  STRUCT
   STAT0 : WORD ;
   STAT1 : WORD ;
   STAT2 : WORD ;
   STAT3 : WORD ;
   STAT4 : WORD ;
   STAT5 : WORD ;
   STAT6 : WORD ;
   STAT7 : WORD ;
   STAT8 : WORD ;
   STAT9 : WORD ;
   STAT10 : WORD ;
   STAT11 : WORD ;
   STAT12 : WORD ;
   STAT13 : WORD ;
   STAT14 : WORD ;
   STAT15 : WORD ;
   STAT16 : INT ;
   STAT17 : INT ;
   STAT18 : INT ;
   STAT19 : INT ;
   STAT20 : ARRAY  [1 .. 6 ] OF BYTE ;
   STAT21 : ARRAY  [1 .. 6 ] OF BYTE ;
   STAT22 : ARRAY  [1 .. 40 ] OF BOOL  := FALSE;
   STAT23 : ARRAY  [1 .. 40 ] OF BOOL  := FALSE;
   STAT24 : WORD ;
   STAT25 : WORD ;
   STAT26 : WORD ;
   STAT27 : WORD ;
   STAT28 : WORD ;
   STAT29 : WORD ;
   STAT30 : WORD ;
   STAT31 : ARRAY  [1 .. 7 ] OF WORD ;
   STAT32 : INT ;
   STAT33 : INT ;
   STAT34 : INT ;
   STAT35 : INT ;
   STAT36 : ARRAY  [1 .. 500 ] OF WORD ;
   STAT37 : ARRAY  [1 .. 16 ] OF BYTE ;
   STAT38 : ARRAY  [1 .. 4 ] OF BYTE ;
   STAT39 : ARRAY  [1 .. 16 ] OF BYTE ;
  END_STRUCT ;
BEGIN
   STAT0 := W#16#0;
   STAT1 := W#16#0;
   STAT2 := W#16#0;
   STAT3 := W#16#0;
   STAT4 := W#16#0;
   STAT5 := W#16#0;
   STAT6 := W#16#0;
   STAT7 := W#16#0;
   STAT8 := W#16#1;
   STAT9 := W#16#9515;
   STAT10 := W#16#2212;
   STAT11 := W#16#8004;
   STAT12 := W#16#1644;
   STAT13 := W#16#0;
   STAT14 := W#16#0;
   STAT15 := W#16#0;
   STAT16 := 0;
   STAT17 := 8;
   STAT18 := 3;
   STAT19 := 0;
   STAT20[1] := B#16#0;
   STAT20[2] := B#16#0;
   STAT20[3] := B#16#0;
   STAT20[4] := B#16#0;
   STAT20[5] := B#16#0;
   STAT20[6] := B#16#0;
   STAT21[1] := B#16#0;
   STAT21[2] := B#16#0;
   STAT21[3] := B#16#0;
   STAT21[4] := B#16#0;
   STAT21[5] := B#16#0;
   STAT21[6] := B#16#0;
   STAT22[1] := FALSE;
   STAT22[2] := FALSE;
   STAT22[3] := TRUE;
   STAT22[4] := FALSE;
   STAT22[5] := FALSE;
   STAT22[6] := FALSE;
   STAT22[7] := FALSE;
   STAT22[8] := TRUE;
   STAT22[9] := FALSE;
   STAT22[10] := FALSE;
   STAT22[11] := FALSE;
   STAT22[12] := FALSE;
   STAT22[13] := FALSE;
   STAT22[14] := FALSE;
   STAT22[15] := FALSE;
   STAT22[16] := FALSE;
   STAT22[17] := FALSE;
   STAT22[18] := FALSE;
   STAT22[19] := FALSE;
   STAT22[20] := FALSE;
   STAT22[21] := FALSE;
   STAT22[22] := FALSE;
   STAT22[23] := FALSE;
   STAT22[24] := FALSE;
   STAT22[25] := FALSE;
   STAT22[26] := FALSE;
   STAT22[27] := FALSE;
   STAT22[28] := FALSE;
   STAT22[29] := FALSE;
   STAT22[30] := FALSE;
   STAT22[31] := FALSE;
   STAT22[32] := FALSE;
   STAT22[33] := FALSE;
   STAT22[34] := FALSE;
   STAT22[35] := FALSE;
   STAT22[36] := FALSE;
   STAT22[37] := FALSE;
   STAT22[38] := FALSE;
   STAT22[39] := FALSE;
   STAT22[40] := FALSE;
   STAT23[1] := FALSE;
   STAT23[2] := FALSE;
   STAT23[3] := FALSE;
   STAT23[4] := FALSE;
   STAT23[5] := FALSE;
   STAT23[6] := TRUE;
   STAT23[7] := FALSE;
   STAT23[8] := FALSE;
   STAT23[9] := FALSE;
   STAT23[10] := FALSE;
   STAT23[11] := FALSE;
   STAT23[12] := FALSE;
   STAT23[13] := FALSE;
   STAT23[14] := FALSE;
   STAT23[15] := FALSE;
   STAT23[16] := FALSE;
   STAT23[17] := FALSE;
   STAT23[18] := FALSE;
   STAT23[19] := FALSE;
   STAT23[20] := FALSE;
   STAT23[21] := FALSE;
   STAT23[22] := FALSE;
   STAT23[23] := FALSE;
   STAT23[24] := FALSE;
   STAT23[25] := TRUE;
   STAT23[26] := FALSE;
   STAT23[27] := FALSE;
   STAT23[28] := FALSE;
   STAT23[29] := FALSE;
   STAT23[30] := FALSE;
   STAT23[31] := FALSE;
   STAT23[32] := FALSE;
   STAT23[33] := FALSE;
   STAT23[34] := FALSE;
   STAT23[35] := FALSE;
   STAT23[36] := FALSE;
   STAT23[37] := FALSE;
   STAT23[38] := FALSE;
   STAT23[39] := FALSE;
   STAT23[40] := FALSE;
   STAT24 := W#16#0;
   STAT25 := W#16#0;
   STAT26 := W#16#0;
   STAT27 := W#16#0;
   STAT28 := W#16#0;
   STAT29 := W#16#0;
   STAT30 := W#16#0;
   STAT31[1] := W#16#0;
   STAT31[2] := W#16#0;
   STAT31[3] := W#16#0;
   STAT31[4] := W#16#0;
   STAT31[5] := W#16#0;
   STAT31[6] := W#16#0;
   STAT31[7] := W#16#0;
   STAT32 := 100;
   STAT33 := 90;
   STAT34 := 80;
   STAT35 := 0;
   STAT36[1] := W#16#600;
   STAT36[2] := W#16#808;
   STAT36[3] := W#16#2930;
   STAT36[4] := W#16#64;
   STAT36[5] := W#16#1;
   STAT36[6] := W#16#600;
   STAT36[7] := W#16#1223;
   STAT36[8] := W#16#4457;
   STAT36[9] := W#16#64;
   STAT36[10] := W#16#9515;
   STAT36[11] := W#16#600;
   STAT36[12] := W#16#908;
   STAT36[13] := W#16#2517;
   STAT36[14] := W#16#64;
   STAT36[15] := W#16#341;
   STAT36[16] := W#16#600;
   STAT36[17] := W#16#522;
   STAT36[18] := W#16#356;
   STAT36[19] := W#16#64;
   STAT36[20] := W#16#8579;
   STAT36[21] := W#16#500;
   STAT36[22] := W#16#1220;
   STAT36[23] := W#16#3131;
   STAT36[24] := W#16#0;
   STAT36[25] := W#16#0;
   STAT36[26] := W#16#0;
   STAT36[27] := W#16#0;
   STAT36[28] := W#16#0;
   STAT36[29] := W#16#0;
   STAT36[30] := W#16#0;
   STAT36[31] := W#16#0;
   STAT36[32] := W#16#0;
   STAT36[33] := W#16#0;
   STAT36[34] := W#16#0;
   STAT36[35] := W#16#0;
   STAT36[36] := W#16#0;
   STAT36[37] := W#16#0;
   STAT36[38] := W#16#0;
   STAT36[39] := W#16#0;
   STAT36[40] := W#16#0;
   STAT36[41] := W#16#0;
   STAT36[42] := W#16#0;
   STAT36[43] := W#16#0;
   STAT36[44] := W#16#0;
   STAT36[45] := W#16#0;
   STAT36[46] := W#16#0;
   STAT36[47] := W#16#0;
   STAT36[48] := W#16#0;
   STAT36[49] := W#16#0;
   STAT36[50] := W#16#0;
   STAT36[51] := W#16#0;
   STAT36[52] := W#16#0;
   STAT36[53] := W#16#0;
   STAT36[54] := W#16#0;
   STAT36[55] := W#16#0;
   STAT36[56] := W#16#0;
   STAT36[57] := W#16#0;
   STAT36[58] := W#16#0;
   STAT36[59] := W#16#0;
   STAT36[60] := W#16#0;
   STAT36[61] := W#16#0;
   STAT36[62] := W#16#0;
   STAT36[63] := W#16#0;
   STAT36[64] := W#16#0;
   STAT36[65] := W#16#0;
   STAT36[66] := W#16#0;
   STAT36[67] := W#16#0;
   STAT36[68] := W#16#0;
   STAT36[69] := W#16#0;
   STAT36[70] := W#16#0;
   STAT36[71] := W#16#0;
   STAT36[72] := W#16#0;
   STAT36[73] := W#16#0;
   STAT36[74] := W#16#0;
   STAT36[75] := W#16#0;
   STAT36[76] := W#16#0;
   STAT36[77] := W#16#0;
   STAT36[78] := W#16#0;
   STAT36[79] := W#16#0;
   STAT36[80] := W#16#0;
   STAT36[81] := W#16#0;
   STAT36[82] := W#16#0;
   STAT36[83] := W#16#0;
   STAT36[84] := W#16#0;
   STAT36[85] := W#16#0;
   STAT36[86] := W#16#0;
   STAT36[87] := W#16#0;
   STAT36[88] := W#16#0;
   STAT36[89] := W#16#0;
   STAT36[90] := W#16#0;
   STAT36[91] := W#16#0;
   STAT36[92] := W#16#0;
   STAT36[93] := W#16#0;
   STAT36[94] := W#16#0;
   STAT36[95] := W#16#0;
   STAT36[96] := W#16#0;
   STAT36[97] := W#16#0;
   STAT36[98] := W#16#0;
   STAT36[99] := W#16#0;
   STAT36[100] := W#16#0;
   STAT36[101] := W#16#0;
   STAT36[102] := W#16#0;
   STAT36[103] := W#16#0;
   STAT36[104] := W#16#0;
   STAT36[105] := W#16#0;
   STAT36[106] := W#16#0;
   STAT36[107] := W#16#0;
   STAT36[108] := W#16#0;
   STAT36[109] := W#16#0;
   STAT36[110] := W#16#0;
   STAT36[111] := W#16#0;
   STAT36[112] := W#16#0;
   STAT36[113] := W#16#0;
   STAT36[114] := W#16#0;
   STAT36[115] := W#16#0;
   STAT36[116] := W#16#0;
   STAT36[117] := W#16#0;
   STAT36[118] := W#16#0;
   STAT36[119] := W#16#0;
   STAT36[120] := W#16#0;
   STAT36[121] := W#16#0;
   STAT36[122] := W#16#0;
   STAT36[123] := W#16#0;
   STAT36[124] := W#16#0;
   STAT36[125] := W#16#0;
   STAT36[126] := W#16#0;
   STAT36[127] := W#16#0;
   STAT36[128] := W#16#0;
   STAT36[129] := W#16#0;
   STAT36[130] := W#16#0;
   STAT36[131] := W#16#0;
   STAT36[132] := W#16#0;
   STAT36[133] := W#16#0;
   STAT36[134] := W#16#0;
   STAT36[135] := W#16#0;
   STAT36[136] := W#16#0;
   STAT36[137] := W#16#0;
   STAT36[138] := W#16#0;
   STAT36[139] := W#16#0;
   STAT36[140] := W#16#0;
   STAT36[141] := W#16#0;
   STAT36[142] := W#16#0;
   STAT36[143] := W#16#0;
   STAT36[144] := W#16#0;
   STAT36[145] := W#16#0;
   STAT36[146] := W#16#0;
   STAT36[147] := W#16#0;
   STAT36[148] := W#16#0;
   STAT36[149] := W#16#0;
   STAT36[150] := W#16#0;
   STAT36[151] := W#16#0;
   STAT36[152] := W#16#0;
   STAT36[153] := W#16#0;
   STAT36[154] := W#16#0;
   STAT36[155] := W#16#0;
   STAT36[156] := W#16#0;
   STAT36[157] := W#16#0;
   STAT36[158] := W#16#0;
   STAT36[159] := W#16#0;
   STAT36[160] := W#16#0;
   STAT36[161] := W#16#0;
   STAT36[162] := W#16#0;
   STAT36[163] := W#16#0;
   STAT36[164] := W#16#0;
   STAT36[165] := W#16#0;
   STAT36[166] := W#16#0;
   STAT36[167] := W#16#0;
   STAT36[168] := W#16#0;
   STAT36[169] := W#16#0;
   STAT36[170] := W#16#0;
   STAT36[171] := W#16#0;
   STAT36[172] := W#16#0;
   STAT36[173] := W#16#0;
   STAT36[174] := W#16#0;
   STAT36[175] := W#16#0;
   STAT36[176] := W#16#0;
   STAT36[177] := W#16#0;
   STAT36[178] := W#16#0;
   STAT36[179] := W#16#0;
   STAT36[180] := W#16#0;
   STAT36[181] := W#16#0;
   STAT36[182] := W#16#0;
   STAT36[183] := W#16#0;
   STAT36[184] := W#16#0;
   STAT36[185] := W#16#0;
   STAT36[186] := W#16#0;
   STAT36[187] := W#16#0;
   STAT36[188] := W#16#0;
   STAT36[189] := W#16#0;
   STAT36[190] := W#16#0;
   STAT36[191] := W#16#0;
   STAT36[192] := W#16#0;
   STAT36[193] := W#16#0;
   STAT36[194] := W#16#0;
   STAT36[195] := W#16#0;
   STAT36[196] := W#16#0;
   STAT36[197] := W#16#0;
   STAT36[198] := W#16#0;
   STAT36[199] := W#16#0;
   STAT36[200] := W#16#0;
   STAT36[201] := W#16#0;
   STAT36[202] := W#16#0;
   STAT36[203] := W#16#0;
   STAT36[204] := W#16#0;
   STAT36[205] := W#16#0;
   STAT36[206] := W#16#0;
   STAT36[207] := W#16#0;
   STAT36[208] := W#16#0;
   STAT36[209] := W#16#0;
   STAT36[210] := W#16#0;
   STAT36[211] := W#16#0;
   STAT36[212] := W#16#0;
   STAT36[213] := W#16#0;
   STAT36[214] := W#16#0;
   STAT36[215] := W#16#0;
   STAT36[216] := W#16#0;
   STAT36[217] := W#16#0;
   STAT36[218] := W#16#0;
   STAT36[219] := W#16#0;
   STAT36[220] := W#16#0;
   STAT36[221] := W#16#0;
   STAT36[222] := W#16#0;
   STAT36[223] := W#16#0;
   STAT36[224] := W#16#0;
   STAT36[225] := W#16#0;
   STAT36[226] := W#16#0;
   STAT36[227] := W#16#0;
   STAT36[228] := W#16#0;
   STAT36[229] := W#16#0;
   STAT36[230] := W#16#0;
   STAT36[231] := W#16#0;
   STAT36[232] := W#16#0;
   STAT36[233] := W#16#0;
   STAT36[234] := W#16#0;
   STAT36[235] := W#16#0;
   STAT36[236] := W#16#0;
   STAT36[237] := W#16#0;
   STAT36[238] := W#16#0;
   STAT36[239] := W#16#0;
   STAT36[240] := W#16#0;
   STAT36[241] := W#16#0;
   STAT36[242] := W#16#0;
   STAT36[243] := W#16#0;
   STAT36[244] := W#16#0;
   STAT36[245] := W#16#0;
   STAT36[246] := W#16#0;
   STAT36[247] := W#16#0;
   STAT36[248] := W#16#0;
   STAT36[249] := W#16#0;
   STAT36[250] := W#16#0;
   STAT36[251] := W#16#0;
   STAT36[252] := W#16#0;
   STAT36[253] := W#16#0;
   STAT36[254] := W#16#0;
   STAT36[255] := W#16#0;
   STAT36[256] := W#16#0;
   STAT36[257] := W#16#0;
   STAT36[258] := W#16#0;
   STAT36[259] := W#16#0;
   STAT36[260] := W#16#0;
   STAT36[261] := W#16#0;
   STAT36[262] := W#16#0;
   STAT36[263] := W#16#0;
   STAT36[264] := W#16#0;
   STAT36[265] := W#16#0;
   STAT36[266] := W#16#0;
   STAT36[267] := W#16#0;
   STAT36[268] := W#16#0;
   STAT36[269] := W#16#0;
   STAT36[270] := W#16#0;
   STAT36[271] := W#16#0;
   STAT36[272] := W#16#0;
   STAT36[273] := W#16#0;
   STAT36[274] := W#16#0;
   STAT36[275] := W#16#0;
   STAT36[276] := W#16#0;
   STAT36[277] := W#16#0;
   STAT36[278] := W#16#0;
   STAT36[279] := W#16#0;
   STAT36[280] := W#16#0;
   STAT36[281] := W#16#0;
   STAT36[282] := W#16#0;
   STAT36[283] := W#16#0;
   STAT36[284] := W#16#0;
   STAT36[285] := W#16#0;
   STAT36[286] := W#16#0;
   STAT36[287] := W#16#0;
   STAT36[288] := W#16#0;
   STAT36[289] := W#16#0;
   STAT36[290] := W#16#0;
   STAT36[291] := W#16#0;
   STAT36[292] := W#16#0;
   STAT36[293] := W#16#0;
   STAT36[294] := W#16#0;
   STAT36[295] := W#16#0;
   STAT36[296] := W#16#0;
   STAT36[297] := W#16#0;
   STAT36[298] := W#16#0;
   STAT36[299] := W#16#0;
   STAT36[300] := W#16#0;
   STAT36[301] := W#16#0;
   STAT36[302] := W#16#0;
   STAT36[303] := W#16#0;
   STAT36[304] := W#16#0;
   STAT36[305] := W#16#0;
   STAT36[306] := W#16#0;
   STAT36[307] := W#16#0;
   STAT36[308] := W#16#0;
   STAT36[309] := W#16#0;
   STAT36[310] := W#16#0;
   STAT36[311] := W#16#0;
   STAT36[312] := W#16#0;
   STAT36[313] := W#16#0;
   STAT36[314] := W#16#0;
   STAT36[315] := W#16#0;
   STAT36[316] := W#16#0;
   STAT36[317] := W#16#0;
   STAT36[318] := W#16#0;
   STAT36[319] := W#16#0;
   STAT36[320] := W#16#0;
   STAT36[321] := W#16#0;
   STAT36[322] := W#16#0;
   STAT36[323] := W#16#0;
   STAT36[324] := W#16#0;
   STAT36[325] := W#16#0;
   STAT36[326] := W#16#0;
   STAT36[327] := W#16#0;
   STAT36[328] := W#16#0;
   STAT36[329] := W#16#0;
   STAT36[330] := W#16#0;
   STAT36[331] := W#16#0;
   STAT36[332] := W#16#0;
   STAT36[333] := W#16#0;
   STAT36[334] := W#16#0;
   STAT36[335] := W#16#0;
   STAT36[336] := W#16#0;
   STAT36[337] := W#16#0;
   STAT36[338] := W#16#0;
   STAT36[339] := W#16#0;
   STAT36[340] := W#16#0;
   STAT36[341] := W#16#0;
   STAT36[342] := W#16#0;
   STAT36[343] := W#16#0;
   STAT36[344] := W#16#0;
   STAT36[345] := W#16#0;
   STAT36[346] := W#16#0;
   STAT36[347] := W#16#0;
   STAT36[348] := W#16#0;
   STAT36[349] := W#16#0;
   STAT36[350] := W#16#0;
   STAT36[351] := W#16#0;
   STAT36[352] := W#16#0;
   STAT36[353] := W#16#0;
   STAT36[354] := W#16#0;
   STAT36[355] := W#16#0;
   STAT36[356] := W#16#0;
   STAT36[357] := W#16#0;
   STAT36[358] := W#16#0;
   STAT36[359] := W#16#0;
   STAT36[360] := W#16#0;
   STAT36[361] := W#16#0;
   STAT36[362] := W#16#0;
   STAT36[363] := W#16#0;
   STAT36[364] := W#16#0;
   STAT36[365] := W#16#0;
   STAT36[366] := W#16#0;
   STAT36[367] := W#16#0;
   STAT36[368] := W#16#0;
   STAT36[369] := W#16#0;
   STAT36[370] := W#16#0;
   STAT36[371] := W#16#0;
   STAT36[372] := W#16#0;
   STAT36[373] := W#16#0;
   STAT36[374] := W#16#0;
   STAT36[375] := W#16#0;
   STAT36[376] := W#16#0;
   STAT36[377] := W#16#0;
   STAT36[378] := W#16#0;
   STAT36[379] := W#16#0;
   STAT36[380] := W#16#0;
   STAT36[381] := W#16#0;
   STAT36[382] := W#16#0;
   STAT36[383] := W#16#0;
   STAT36[384] := W#16#0;
   STAT36[385] := W#16#0;
   STAT36[386] := W#16#0;
   STAT36[387] := W#16#0;
   STAT36[388] := W#16#0;
   STAT36[389] := W#16#0;
   STAT36[390] := W#16#0;
   STAT36[391] := W#16#0;
   STAT36[392] := W#16#0;
   STAT36[393] := W#16#0;
   STAT36[394] := W#16#0;
   STAT36[395] := W#16#0;
   STAT36[396] := W#16#0;
   STAT36[397] := W#16#0;
   STAT36[398] := W#16#0;
   STAT36[399] := W#16#0;
   STAT36[400] := W#16#0;
   STAT36[401] := W#16#0;
   STAT36[402] := W#16#0;
   STAT36[403] := W#16#0;
   STAT36[404] := W#16#0;
   STAT36[405] := W#16#0;
   STAT36[406] := W#16#0;
   STAT36[407] := W#16#0;
   STAT36[408] := W#16#0;
   STAT36[409] := W#16#0;
   STAT36[410] := W#16#0;
   STAT36[411] := W#16#0;
   STAT36[412] := W#16#0;
   STAT36[413] := W#16#0;
   STAT36[414] := W#16#0;
   STAT36[415] := W#16#0;
   STAT36[416] := W#16#0;
   STAT36[417] := W#16#0;
   STAT36[418] := W#16#0;
   STAT36[419] := W#16#0;
   STAT36[420] := W#16#0;
   STAT36[421] := W#16#0;
   STAT36[422] := W#16#0;
   STAT36[423] := W#16#0;
   STAT36[424] := W#16#0;
   STAT36[425] := W#16#0;
   STAT36[426] := W#16#0;
   STAT36[427] := W#16#0;
   STAT36[428] := W#16#0;
   STAT36[429] := W#16#0;
   STAT36[430] := W#16#0;
   STAT36[431] := W#16#0;
   STAT36[432] := W#16#0;
   STAT36[433] := W#16#0;
   STAT36[434] := W#16#0;
   STAT36[435] := W#16#0;
   STAT36[436] := W#16#0;
   STAT36[437] := W#16#0;
   STAT36[438] := W#16#0;
   STAT36[439] := W#16#0;
   STAT36[440] := W#16#0;
   STAT36[441] := W#16#0;
   STAT36[442] := W#16#0;
   STAT36[443] := W#16#0;
   STAT36[444] := W#16#0;
   STAT36[445] := W#16#0;
   STAT36[446] := W#16#0;
   STAT36[447] := W#16#0;
   STAT36[448] := W#16#0;
   STAT36[449] := W#16#0;
   STAT36[450] := W#16#0;
   STAT36[451] := W#16#0;
   STAT36[452] := W#16#0;
   STAT36[453] := W#16#0;
   STAT36[454] := W#16#0;
   STAT36[455] := W#16#0;
   STAT36[456] := W#16#0;
   STAT36[457] := W#16#0;
   STAT36[458] := W#16#0;
   STAT36[459] := W#16#0;
   STAT36[460] := W#16#0;
   STAT36[461] := W#16#0;
   STAT36[462] := W#16#0;
   STAT36[463] := W#16#0;
   STAT36[464] := W#16#0;
   STAT36[465] := W#16#0;
   STAT36[466] := W#16#0;
   STAT36[467] := W#16#0;
   STAT36[468] := W#16#0;
   STAT36[469] := W#16#0;
   STAT36[470] := W#16#0;
   STAT36[471] := W#16#0;
   STAT36[472] := W#16#0;
   STAT36[473] := W#16#0;
   STAT36[474] := W#16#0;
   STAT36[475] := W#16#0;
   STAT36[476] := W#16#0;
   STAT36[477] := W#16#0;
   STAT36[478] := W#16#0;
   STAT36[479] := W#16#0;
   STAT36[480] := W#16#0;
   STAT36[481] := W#16#0;
   STAT36[482] := W#16#0;
   STAT36[483] := W#16#0;
   STAT36[484] := W#16#0;
   STAT36[485] := W#16#0;
   STAT36[486] := W#16#0;
   STAT36[487] := W#16#0;
   STAT36[488] := W#16#0;
   STAT36[489] := W#16#0;
   STAT36[490] := W#16#0;
   STAT36[491] := W#16#0;
   STAT36[492] := W#16#0;
   STAT36[493] := W#16#0;
   STAT36[494] := W#16#0;
   STAT36[495] := W#16#0;
   STAT36[496] := W#16#0;
   STAT36[497] := W#16#0;
   STAT36[498] := W#16#0;
   STAT36[499] := W#16#0;
   STAT36[500] := W#16#0;
   STAT37[1] := B#16#0;
   STAT37[2] := B#16#0;
   STAT37[3] := B#16#0;
   STAT37[4] := B#16#1;
   STAT37[5] := B#16#22;
   STAT37[6] := B#16#42;
   STAT37[7] := B#16#80;
   STAT37[8] := B#16#80;
   STAT37[9] := B#16#26;
   STAT37[10] := B#16#10;
   STAT37[11] := B#16#0;
   STAT37[12] := B#16#0;
   STAT37[13] := B#16#0;
   STAT37[14] := B#16#0;
   STAT37[15] := B#16#0;
   STAT37[16] := B#16#0;
   STAT38[1] := B#16#0;
   STAT38[2] := B#16#0;
   STAT38[3] := B#16#0;
   STAT38[4] := B#16#0;
   STAT39[1] := B#16#95;
   STAT39[2] := B#16#15;
   STAT39[3] := B#16#0;
   STAT39[4] := B#16#1;
   STAT39[5] := B#16#12;
   STAT39[6] := B#16#22;
   STAT39[7] := B#16#4;
   STAT39[8] := B#16#80;
   STAT39[9] := B#16#44;
   STAT39[10] := B#16#16;
   STAT39[11] := B#16#0;
   STAT39[12] := B#16#0;
   STAT39[13] := B#16#0;
   STAT39[14] := B#16#0;
   STAT39[15] := B#16#0;
   STAT39[16] := B#16#0;
END_DATA_BLOCK

DATA_BLOCK DB 164
VERSION : 0.1


  STRUCT
   STAT0 : WORD ;
   STAT1 : WORD ;
   STAT2 : WORD ;
   STAT3 : WORD ;
   STAT4 : WORD ;
   STAT5 : WORD ;
   STAT6 : WORD ;
   STAT7 : WORD ;
   STAT8 : WORD ;
   STAT9 : WORD ;
   STAT10 : WORD ;
   STAT11 : WORD ;
   STAT12 : WORD ;
   STAT13 : WORD ;
   STAT14 : WORD ;
   STAT15 : WORD ;
   STAT16 : INT ;
   STAT17 : INT ;
   STAT18 : INT ;
   STAT19 : INT ;
   STAT20 : ARRAY  [1 .. 6 ] OF BYTE ;
   STAT21 : ARRAY  [1 .. 6 ] OF BYTE ;
   STAT22 : ARRAY  [1 .. 40 ] OF BOOL  := FALSE;
   STAT23 : ARRAY  [1 .. 40 ] OF BOOL  := FALSE;
   STAT24 : WORD ;
   STAT25 : WORD ;
   STAT26 : WORD ;
   STAT27 : WORD ;
   STAT28 : WORD ;
   STAT29 : WORD ;
   STAT30 : WORD ;
   STAT31 : ARRAY  [1 .. 7 ] OF WORD ;
   STAT32 : INT ;
   STAT33 : INT ;
   STAT34 : INT ;
   STAT35 : INT ;
   STAT36 : ARRAY  [1 .. 500 ] OF WORD ;
   STAT37 : ARRAY  [1 .. 16 ] OF BYTE ;
   STAT38 : ARRAY  [1 .. 4 ] OF BYTE ;
   STAT39 : ARRAY  [1 .. 16 ] OF BYTE ;
  END_STRUCT ;
BEGIN
   STAT0 := W#16#0;
   STAT1 := W#16#0;
   STAT2 := W#16#0;
   STAT3 := W#16#0;
   STAT4 := W#16#0;
   STAT5 := W#16#0;
   STAT6 := W#16#0;
   STAT7 := W#16#0;
   STAT8 := W#16#0;
   STAT9 := W#16#0;
   STAT10 := W#16#0;
   STAT11 := W#16#0;
   STAT12 := W#16#0;
   STAT13 := W#16#0;
   STAT14 := W#16#0;
   STAT15 := W#16#0;
   STAT16 := 0;
   STAT17 := 10;
   STAT18 := 3;
   STAT19 := 0;
   STAT20[1] := B#16#0;
   STAT20[2] := B#16#0;
   STAT20[3] := B#16#0;
   STAT20[4] := B#16#0;
   STAT20[5] := B#16#0;
   STAT20[6] := B#16#0;
   STAT21[1] := B#16#0;
   STAT21[2] := B#16#0;
   STAT21[3] := B#16#0;
   STAT21[4] := B#16#0;
   STAT21[5] := B#16#0;
   STAT21[6] := B#16#0;
   STAT22[1] := FALSE;
   STAT22[2] := FALSE;
   STAT22[3] := TRUE;
   STAT22[4] := FALSE;
   STAT22[5] := FALSE;
   STAT22[6] := FALSE;
   STAT22[7] := FALSE;
   STAT22[8] := TRUE;
   STAT22[9] := FALSE;
   STAT22[10] := FALSE;
   STAT22[11] := FALSE;
   STAT22[12] := FALSE;
   STAT22[13] := FALSE;
   STAT22[14] := FALSE;
   STAT22[15] := FALSE;
   STAT22[16] := FALSE;
   STAT22[17] := FALSE;
   STAT22[18] := FALSE;
   STAT22[19] := FALSE;
   STAT22[20] := FALSE;
   STAT22[21] := FALSE;
   STAT22[22] := FALSE;
   STAT22[23] := FALSE;
   STAT22[24] := FALSE;
   STAT22[25] := FALSE;
   STAT22[26] := FALSE;
   STAT22[27] := FALSE;
   STAT22[28] := FALSE;
   STAT22[29] := FALSE;
   STAT22[30] := FALSE;
   STAT22[31] := FALSE;
   STAT22[32] := FALSE;
   STAT22[33] := FALSE;
   STAT22[34] := FALSE;
   STAT22[35] := FALSE;
   STAT22[36] := FALSE;
   STAT22[37] := FALSE;
   STAT22[38] := FALSE;
   STAT22[39] := FALSE;
   STAT22[40] := FALSE;
   STAT23[1] := FALSE;
   STAT23[2] := FALSE;
   STAT23[3] := FALSE;
   STAT23[4] := FALSE;
   STAT23[5] := FALSE;
   STAT23[6] := TRUE;
   STAT23[7] := FALSE;
   STAT23[8] := FALSE;
   STAT23[9] := FALSE;
   STAT23[10] := FALSE;
   STAT23[11] := FALSE;
   STAT23[12] := FALSE;
   STAT23[13] := FALSE;
   STAT23[14] := FALSE;
   STAT23[15] := FALSE;
   STAT23[16] := FALSE;
   STAT23[17] := FALSE;
   STAT23[18] := FALSE;
   STAT23[19] := FALSE;
   STAT23[20] := FALSE;
   STAT23[21] := FALSE;
   STAT23[22] := FALSE;
   STAT23[23] := FALSE;
   STAT23[24] := FALSE;
   STAT23[25] := TRUE;
   STAT23[26] := FALSE;
   STAT23[27] := FALSE;
   STAT23[28] := FALSE;
   STAT23[29] := FALSE;
   STAT23[30] := FALSE;
   STAT23[31] := FALSE;
   STAT23[32] := FALSE;
   STAT23[33] := FALSE;
   STAT23[34] := FALSE;
   STAT23[35] := FALSE;
   STAT23[36] := FALSE;
   STAT23[37] := FALSE;
   STAT23[38] := FALSE;
   STAT23[39] := FALSE;
   STAT23[40] := FALSE;
   STAT24 := W#16#0;
   STAT25 := W#16#0;
   STAT26 := W#16#0;
   STAT27 := W#16#0;
   STAT28 := W#16#0;
   STAT29 := W#16#0;
   STAT30 := W#16#0;
   STAT31[1] := W#16#0;
   STAT31[2] := W#16#0;
   STAT31[3] := W#16#0;
   STAT31[4] := W#16#0;
   STAT31[5] := W#16#0;
   STAT31[6] := W#16#0;
   STAT31[7] := W#16#0;
   STAT32 := 100;
   STAT33 := 90;
   STAT34 := 80;
   STAT35 := 0;
   STAT36[1] := W#16#600;
   STAT36[2] := W#16#2113;
   STAT36[3] := W#16#858;
   STAT36[4] := W#16#64;
   STAT36[5] := W#16#7925;
   STAT36[6] := W#16#600;
   STAT36[7] := W#16#1420;
   STAT36[8] := W#16#2809;
   STAT36[9] := W#16#64;
   STAT36[10] := W#16#1592;
   STAT36[11] := W#16#600;
   STAT36[12] := W#16#1414;
   STAT36[13] := W#16#205;
   STAT36[14] := W#16#64;
   STAT36[15] := W#16#1592;
   STAT36[16] := W#16#600;
   STAT36[17] := W#16#616;
   STAT36[18] := W#16#1124;
   STAT36[19] := W#16#64;
   STAT36[20] := W#16#3330;
   STAT36[21] := W#16#600;
   STAT36[22] := W#16#1310;
   STAT36[23] := W#16#2206;
   STAT36[24] := W#16#64;
   STAT36[25] := W#16#575;
   STAT36[26] := W#16#500;
   STAT36[27] := W#16#1220;
   STAT36[28] := W#16#3131;
   STAT36[29] := W#16#0;
   STAT36[30] := W#16#0;
   STAT36[31] := W#16#0;
   STAT36[32] := W#16#0;
   STAT36[33] := W#16#0;
   STAT36[34] := W#16#0;
   STAT36[35] := W#16#0;
   STAT36[36] := W#16#0;
   STAT36[37] := W#16#0;
   STAT36[38] := W#16#0;
   STAT36[39] := W#16#0;
   STAT36[40] := W#16#0;
   STAT36[41] := W#16#0;
   STAT36[42] := W#16#0;
   STAT36[43] := W#16#0;
   STAT36[44] := W#16#0;
   STAT36[45] := W#16#0;
   STAT36[46] := W#16#0;
   STAT36[47] := W#16#0;
   STAT36[48] := W#16#0;
   STAT36[49] := W#16#0;
   STAT36[50] := W#16#0;
   STAT36[51] := W#16#0;
   STAT36[52] := W#16#0;
   STAT36[53] := W#16#0;
   STAT36[54] := W#16#0;
   STAT36[55] := W#16#0;
   STAT36[56] := W#16#0;
   STAT36[57] := W#16#0;
   STAT36[58] := W#16#0;
   STAT36[59] := W#16#0;
   STAT36[60] := W#16#0;
   STAT36[61] := W#16#0;
   STAT36[62] := W#16#0;
   STAT36[63] := W#16#0;
   STAT36[64] := W#16#0;
   STAT36[65] := W#16#0;
   STAT36[66] := W#16#0;
   STAT36[67] := W#16#0;
   STAT36[68] := W#16#0;
   STAT36[69] := W#16#0;
   STAT36[70] := W#16#0;
   STAT36[71] := W#16#0;
   STAT36[72] := W#16#0;
   STAT36[73] := W#16#0;
   STAT36[74] := W#16#0;
   STAT36[75] := W#16#0;
   STAT36[76] := W#16#0;
   STAT36[77] := W#16#0;
   STAT36[78] := W#16#0;
   STAT36[79] := W#16#0;
   STAT36[80] := W#16#0;
   STAT36[81] := W#16#0;
   STAT36[82] := W#16#0;
   STAT36[83] := W#16#0;
   STAT36[84] := W#16#0;
   STAT36[85] := W#16#0;
   STAT36[86] := W#16#0;
   STAT36[87] := W#16#0;
   STAT36[88] := W#16#0;
   STAT36[89] := W#16#0;
   STAT36[90] := W#16#0;
   STAT36[91] := W#16#0;
   STAT36[92] := W#16#0;
   STAT36[93] := W#16#0;
   STAT36[94] := W#16#0;
   STAT36[95] := W#16#0;
   STAT36[96] := W#16#0;
   STAT36[97] := W#16#0;
   STAT36[98] := W#16#0;
   STAT36[99] := W#16#0;
   STAT36[100] := W#16#0;
   STAT36[101] := W#16#0;
   STAT36[102] := W#16#0;
   STAT36[103] := W#16#0;
   STAT36[104] := W#16#0;
   STAT36[105] := W#16#0;
   STAT36[106] := W#16#0;
   STAT36[107] := W#16#0;
   STAT36[108] := W#16#0;
   STAT36[109] := W#16#0;
   STAT36[110] := W#16#0;
   STAT36[111] := W#16#0;
   STAT36[112] := W#16#0;
   STAT36[113] := W#16#0;
   STAT36[114] := W#16#0;
   STAT36[115] := W#16#0;
   STAT36[116] := W#16#0;
   STAT36[117] := W#16#0;
   STAT36[118] := W#16#0;
   STAT36[119] := W#16#0;
   STAT36[120] := W#16#0;
   STAT36[121] := W#16#0;
   STAT36[122] := W#16#0;
   STAT36[123] := W#16#0;
   STAT36[124] := W#16#0;
   STAT36[125] := W#16#0;
   STAT36[126] := W#16#0;
   STAT36[127] := W#16#0;
   STAT36[128] := W#16#0;
   STAT36[129] := W#16#0;
   STAT36[130] := W#16#0;
   STAT36[131] := W#16#0;
   STAT36[132] := W#16#0;
   STAT36[133] := W#16#0;
   STAT36[134] := W#16#0;
   STAT36[135] := W#16#0;
   STAT36[136] := W#16#0;
   STAT36[137] := W#16#0;
   STAT36[138] := W#16#0;
   STAT36[139] := W#16#0;
   STAT36[140] := W#16#0;
   STAT36[141] := W#16#0;
   STAT36[142] := W#16#0;
   STAT36[143] := W#16#0;
   STAT36[144] := W#16#0;
   STAT36[145] := W#16#0;
   STAT36[146] := W#16#0;
   STAT36[147] := W#16#0;
   STAT36[148] := W#16#0;
   STAT36[149] := W#16#0;
   STAT36[150] := W#16#0;
   STAT36[151] := W#16#0;
   STAT36[152] := W#16#0;
   STAT36[153] := W#16#0;
   STAT36[154] := W#16#0;
   STAT36[155] := W#16#0;
   STAT36[156] := W#16#0;
   STAT36[157] := W#16#0;
   STAT36[158] := W#16#0;
   STAT36[159] := W#16#0;
   STAT36[160] := W#16#0;
   STAT36[161] := W#16#0;
   STAT36[162] := W#16#0;
   STAT36[163] := W#16#0;
   STAT36[164] := W#16#0;
   STAT36[165] := W#16#0;
   STAT36[166] := W#16#0;
   STAT36[167] := W#16#0;
   STAT36[168] := W#16#0;
   STAT36[169] := W#16#0;
   STAT36[170] := W#16#0;
   STAT36[171] := W#16#0;
   STAT36[172] := W#16#0;
   STAT36[173] := W#16#0;
   STAT36[174] := W#16#0;
   STAT36[175] := W#16#0;
   STAT36[176] := W#16#0;
   STAT36[177] := W#16#0;
   STAT36[178] := W#16#0;
   STAT36[179] := W#16#0;
   STAT36[180] := W#16#0;
   STAT36[181] := W#16#0;
   STAT36[182] := W#16#0;
   STAT36[183] := W#16#0;
   STAT36[184] := W#16#0;
   STAT36[185] := W#16#0;
   STAT36[186] := W#16#0;
   STAT36[187] := W#16#0;
   STAT36[188] := W#16#0;
   STAT36[189] := W#16#0;
   STAT36[190] := W#16#0;
   STAT36[191] := W#16#0;
   STAT36[192] := W#16#0;
   STAT36[193] := W#16#0;
   STAT36[194] := W#16#0;
   STAT36[195] := W#16#0;
   STAT36[196] := W#16#0;
   STAT36[197] := W#16#0;
   STAT36[198] := W#16#0;
   STAT36[199] := W#16#0;
   STAT36[200] := W#16#0;
   STAT36[201] := W#16#0;
   STAT36[202] := W#16#0;
   STAT36[203] := W#16#0;
   STAT36[204] := W#16#0;
   STAT36[205] := W#16#0;
   STAT36[206] := W#16#0;
   STAT36[207] := W#16#0;
   STAT36[208] := W#16#0;
   STAT36[209] := W#16#0;
   STAT36[210] := W#16#0;
   STAT36[211] := W#16#0;
   STAT36[212] := W#16#0;
   STAT36[213] := W#16#0;
   STAT36[214] := W#16#0;
   STAT36[215] := W#16#0;
   STAT36[216] := W#16#0;
   STAT36[217] := W#16#0;
   STAT36[218] := W#16#0;
   STAT36[219] := W#16#0;
   STAT36[220] := W#16#0;
   STAT36[221] := W#16#0;
   STAT36[222] := W#16#0;
   STAT36[223] := W#16#0;
   STAT36[224] := W#16#0;
   STAT36[225] := W#16#0;
   STAT36[226] := W#16#0;
   STAT36[227] := W#16#0;
   STAT36[228] := W#16#0;
   STAT36[229] := W#16#0;
   STAT36[230] := W#16#0;
   STAT36[231] := W#16#0;
   STAT36[232] := W#16#0;
   STAT36[233] := W#16#0;
   STAT36[234] := W#16#0;
   STAT36[235] := W#16#0;
   STAT36[236] := W#16#0;
   STAT36[237] := W#16#0;
   STAT36[238] := W#16#0;
   STAT36[239] := W#16#0;
   STAT36[240] := W#16#0;
   STAT36[241] := W#16#0;
   STAT36[242] := W#16#0;
   STAT36[243] := W#16#0;
   STAT36[244] := W#16#0;
   STAT36[245] := W#16#0;
   STAT36[246] := W#16#0;
   STAT36[247] := W#16#0;
   STAT36[248] := W#16#0;
   STAT36[249] := W#16#0;
   STAT36[250] := W#16#0;
   STAT36[251] := W#16#0;
   STAT36[252] := W#16#0;
   STAT36[253] := W#16#0;
   STAT36[254] := W#16#0;
   STAT36[255] := W#16#0;
   STAT36[256] := W#16#0;
   STAT36[257] := W#16#0;
   STAT36[258] := W#16#0;
   STAT36[259] := W#16#0;
   STAT36[260] := W#16#0;
   STAT36[261] := W#16#0;
   STAT36[262] := W#16#0;
   STAT36[263] := W#16#0;
   STAT36[264] := W#16#0;
   STAT36[265] := W#16#0;
   STAT36[266] := W#16#0;
   STAT36[267] := W#16#0;
   STAT36[268] := W#16#0;
   STAT36[269] := W#16#0;
   STAT36[270] := W#16#0;
   STAT36[271] := W#16#0;
   STAT36[272] := W#16#0;
   STAT36[273] := W#16#0;
   STAT36[274] := W#16#0;
   STAT36[275] := W#16#0;
   STAT36[276] := W#16#0;
   STAT36[277] := W#16#0;
   STAT36[278] := W#16#0;
   STAT36[279] := W#16#0;
   STAT36[280] := W#16#0;
   STAT36[281] := W#16#0;
   STAT36[282] := W#16#0;
   STAT36[283] := W#16#0;
   STAT36[284] := W#16#0;
   STAT36[285] := W#16#0;
   STAT36[286] := W#16#0;
   STAT36[287] := W#16#0;
   STAT36[288] := W#16#0;
   STAT36[289] := W#16#0;
   STAT36[290] := W#16#0;
   STAT36[291] := W#16#0;
   STAT36[292] := W#16#0;
   STAT36[293] := W#16#0;
   STAT36[294] := W#16#0;
   STAT36[295] := W#16#0;
   STAT36[296] := W#16#0;
   STAT36[297] := W#16#0;
   STAT36[298] := W#16#0;
   STAT36[299] := W#16#0;
   STAT36[300] := W#16#0;
   STAT36[301] := W#16#0;
   STAT36[302] := W#16#0;
   STAT36[303] := W#16#0;
   STAT36[304] := W#16#0;
   STAT36[305] := W#16#0;
   STAT36[306] := W#16#0;
   STAT36[307] := W#16#0;
   STAT36[308] := W#16#0;
   STAT36[309] := W#16#0;
   STAT36[310] := W#16#0;
   STAT36[311] := W#16#0;
   STAT36[312] := W#16#0;
   STAT36[313] := W#16#0;
   STAT36[314] := W#16#0;
   STAT36[315] := W#16#0;
   STAT36[316] := W#16#0;
   STAT36[317] := W#16#0;
   STAT36[318] := W#16#0;
   STAT36[319] := W#16#0;
   STAT36[320] := W#16#0;
   STAT36[321] := W#16#0;
   STAT36[322] := W#16#0;
   STAT36[323] := W#16#0;
   STAT36[324] := W#16#0;
   STAT36[325] := W#16#0;
   STAT36[326] := W#16#0;
   STAT36[327] := W#16#0;
   STAT36[328] := W#16#0;
   STAT36[329] := W#16#0;
   STAT36[330] := W#16#0;
   STAT36[331] := W#16#0;
   STAT36[332] := W#16#0;
   STAT36[333] := W#16#0;
   STAT36[334] := W#16#0;
   STAT36[335] := W#16#0;
   STAT36[336] := W#16#0;
   STAT36[337] := W#16#0;
   STAT36[338] := W#16#0;
   STAT36[339] := W#16#0;
   STAT36[340] := W#16#0;
   STAT36[341] := W#16#0;
   STAT36[342] := W#16#0;
   STAT36[343] := W#16#0;
   STAT36[344] := W#16#0;
   STAT36[345] := W#16#0;
   STAT36[346] := W#16#0;
   STAT36[347] := W#16#0;
   STAT36[348] := W#16#0;
   STAT36[349] := W#16#0;
   STAT36[350] := W#16#0;
   STAT36[351] := W#16#0;
   STAT36[352] := W#16#0;
   STAT36[353] := W#16#0;
   STAT36[354] := W#16#0;
   STAT36[355] := W#16#0;
   STAT36[356] := W#16#0;
   STAT36[357] := W#16#0;
   STAT36[358] := W#16#0;
   STAT36[359] := W#16#0;
   STAT36[360] := W#16#0;
   STAT36[361] := W#16#0;
   STAT36[362] := W#16#0;
   STAT36[363] := W#16#0;
   STAT36[364] := W#16#0;
   STAT36[365] := W#16#0;
   STAT36[366] := W#16#0;
   STAT36[367] := W#16#0;
   STAT36[368] := W#16#0;
   STAT36[369] := W#16#0;
   STAT36[370] := W#16#0;
   STAT36[371] := W#16#0;
   STAT36[372] := W#16#0;
   STAT36[373] := W#16#0;
   STAT36[374] := W#16#0;
   STAT36[375] := W#16#0;
   STAT36[376] := W#16#0;
   STAT36[377] := W#16#0;
   STAT36[378] := W#16#0;
   STAT36[379] := W#16#0;
   STAT36[380] := W#16#0;
   STAT36[381] := W#16#0;
   STAT36[382] := W#16#0;
   STAT36[383] := W#16#0;
   STAT36[384] := W#16#0;
   STAT36[385] := W#16#0;
   STAT36[386] := W#16#0;
   STAT36[387] := W#16#0;
   STAT36[388] := W#16#0;
   STAT36[389] := W#16#0;
   STAT36[390] := W#16#0;
   STAT36[391] := W#16#0;
   STAT36[392] := W#16#0;
   STAT36[393] := W#16#0;
   STAT36[394] := W#16#0;
   STAT36[395] := W#16#0;
   STAT36[396] := W#16#0;
   STAT36[397] := W#16#0;
   STAT36[398] := W#16#0;
   STAT36[399] := W#16#0;
   STAT36[400] := W#16#0;
   STAT36[401] := W#16#0;
   STAT36[402] := W#16#0;
   STAT36[403] := W#16#0;
   STAT36[404] := W#16#0;
   STAT36[405] := W#16#0;
   STAT36[406] := W#16#0;
   STAT36[407] := W#16#0;
   STAT36[408] := W#16#0;
   STAT36[409] := W#16#0;
   STAT36[410] := W#16#0;
   STAT36[411] := W#16#0;
   STAT36[412] := W#16#0;
   STAT36[413] := W#16#0;
   STAT36[414] := W#16#0;
   STAT36[415] := W#16#0;
   STAT36[416] := W#16#0;
   STAT36[417] := W#16#0;
   STAT36[418] := W#16#0;
   STAT36[419] := W#16#0;
   STAT36[420] := W#16#0;
   STAT36[421] := W#16#0;
   STAT36[422] := W#16#0;
   STAT36[423] := W#16#0;
   STAT36[424] := W#16#0;
   STAT36[425] := W#16#0;
   STAT36[426] := W#16#0;
   STAT36[427] := W#16#0;
   STAT36[428] := W#16#0;
   STAT36[429] := W#16#0;
   STAT36[430] := W#16#0;
   STAT36[431] := W#16#0;
   STAT36[432] := W#16#0;
   STAT36[433] := W#16#0;
   STAT36[434] := W#16#0;
   STAT36[435] := W#16#0;
   STAT36[436] := W#16#0;
   STAT36[437] := W#16#0;
   STAT36[438] := W#16#0;
   STAT36[439] := W#16#0;
   STAT36[440] := W#16#0;
   STAT36[441] := W#16#0;
   STAT36[442] := W#16#0;
   STAT36[443] := W#16#0;
   STAT36[444] := W#16#0;
   STAT36[445] := W#16#0;
   STAT36[446] := W#16#0;
   STAT36[447] := W#16#0;
   STAT36[448] := W#16#0;
   STAT36[449] := W#16#0;
   STAT36[450] := W#16#0;
   STAT36[451] := W#16#0;
   STAT36[452] := W#16#0;
   STAT36[453] := W#16#0;
   STAT36[454] := W#16#0;
   STAT36[455] := W#16#0;
   STAT36[456] := W#16#0;
   STAT36[457] := W#16#0;
   STAT36[458] := W#16#0;
   STAT36[459] := W#16#0;
   STAT36[460] := W#16#0;
   STAT36[461] := W#16#0;
   STAT36[462] := W#16#0;
   STAT36[463] := W#16#0;
   STAT36[464] := W#16#0;
   STAT36[465] := W#16#0;
   STAT36[466] := W#16#0;
   STAT36[467] := W#16#0;
   STAT36[468] := W#16#0;
   STAT36[469] := W#16#0;
   STAT36[470] := W#16#0;
   STAT36[471] := W#16#0;
   STAT36[472] := W#16#0;
   STAT36[473] := W#16#0;
   STAT36[474] := W#16#0;
   STAT36[475] := W#16#0;
   STAT36[476] := W#16#0;
   STAT36[477] := W#16#0;
   STAT36[478] := W#16#0;
   STAT36[479] := W#16#0;
   STAT36[480] := W#16#0;
   STAT36[481] := W#16#0;
   STAT36[482] := W#16#0;
   STAT36[483] := W#16#0;
   STAT36[484] := W#16#0;
   STAT36[485] := W#16#0;
   STAT36[486] := W#16#0;
   STAT36[487] := W#16#0;
   STAT36[488] := W#16#0;
   STAT36[489] := W#16#0;
   STAT36[490] := W#16#0;
   STAT36[491] := W#16#0;
   STAT36[492] := W#16#0;
   STAT36[493] := W#16#0;
   STAT36[494] := W#16#0;
   STAT36[495] := W#16#0;
   STAT36[496] := W#16#0;
   STAT36[497] := W#16#0;
   STAT36[498] := W#16#0;
   STAT36[499] := W#16#0;
   STAT36[500] := W#16#0;
   STAT37[1] := B#16#0;
   STAT37[2] := B#16#13;
   STAT37[3] := B#16#79;
   STAT37[4] := B#16#25;
   STAT37[5] := B#16#21;
   STAT37[6] := B#16#2;
   STAT37[7] := B#16#81;
   STAT37[8] := B#16#4;
   STAT37[9] := B#16#16;
   STAT37[10] := B#16#54;
   STAT37[11] := B#16#0;
   STAT37[12] := B#16#0;
   STAT37[13] := B#16#0;
   STAT37[14] := B#16#0;
   STAT37[15] := B#16#0;
   STAT37[16] := B#16#0;
   STAT38[1] := B#16#0;
   STAT38[2] := B#16#0;
   STAT38[3] := B#16#0;
   STAT38[4] := B#16#0;
   STAT39[1] := B#16#0;
   STAT39[2] := B#16#0;
   STAT39[3] := B#16#0;
   STAT39[4] := B#16#0;
   STAT39[5] := B#16#0;
   STAT39[6] := B#16#0;
   STAT39[7] := B#16#0;
   STAT39[8] := B#16#0;
   STAT39[9] := B#16#0;
   STAT39[10] := B#16#0;
   STAT39[11] := B#16#0;
   STAT39[12] := B#16#0;
   STAT39[13] := B#16#0;
   STAT39[14] := B#16#0;
   STAT39[15] := B#16#0;
   STAT39[16] := B#16#0;
END_DATA_BLOCK

DATA_BLOCK DB 165
VERSION : 0.1


  STRUCT
   STAT0 : WORD ;
   STAT1 : WORD ;
   STAT2 : WORD ;
   STAT3 : WORD ;
   STAT4 : WORD ;
   STAT5 : WORD ;
   STAT6 : WORD ;
   STAT7 : WORD ;
   STAT8 : WORD ;
   STAT9 : WORD ;
   STAT10 : WORD ;
   STAT11 : WORD ;
   STAT12 : WORD ;
   STAT13 : WORD ;
   STAT14 : WORD ;
   STAT15 : WORD ;
   STAT16 : INT ;
   STAT17 : INT ;
   STAT18 : INT ;
   STAT19 : INT ;
   STAT20 : ARRAY  [1 .. 6 ] OF BYTE ;
   STAT21 : ARRAY  [1 .. 6 ] OF BYTE ;
   STAT22 : ARRAY  [1 .. 40 ] OF BOOL  := FALSE;
   STAT23 : ARRAY  [1 .. 40 ] OF BOOL  := FALSE;
   STAT24 : WORD ;
   STAT25 : WORD ;
   STAT26 : WORD ;
   STAT27 : WORD ;
   STAT28 : WORD ;
   STAT29 : WORD ;
   STAT30 : WORD ;
   STAT31 : ARRAY  [1 .. 7 ] OF WORD ;
   STAT32 : INT ;
   STAT33 : INT ;
   STAT34 : INT ;
   STAT35 : INT ;
   STAT36 : ARRAY  [1 .. 500 ] OF WORD ;
   STAT37 : ARRAY  [1 .. 16 ] OF BYTE ;
   STAT38 : ARRAY  [1 .. 4 ] OF BYTE ;
   STAT39 : ARRAY  [1 .. 16 ] OF BYTE ;
  END_STRUCT ;
BEGIN
   STAT0 := W#16#2717;
   STAT1 := W#16#87;
   STAT2 := W#16#A22;
   STAT3 := W#16#1080;
   STAT4 := W#16#5416;
   STAT5 := W#16#40;
   STAT6 := W#16#0;
   STAT7 := W#16#0;
   STAT8 := W#16#87;
   STAT9 := W#16#2716;
   STAT10 := W#16#2222;
   STAT11 := W#16#8004;
   STAT12 := W#16#1610;
   STAT13 := W#16#6000;
   STAT14 := W#16#0;
   STAT15 := W#16#0;
   STAT16 := 0;
   STAT17 := 4;
   STAT18 := 3;
   STAT19 := 0;
   STAT20[1] := B#16#0;
   STAT20[2] := B#16#0;
   STAT20[3] := B#16#0;
   STAT20[4] := B#16#0;
   STAT20[5] := B#16#0;
   STAT20[6] := B#16#0;
   STAT21[1] := B#16#0;
   STAT21[2] := B#16#0;
   STAT21[3] := B#16#0;
   STAT21[4] := B#16#0;
   STAT21[5] := B#16#0;
   STAT21[6] := B#16#0;
   STAT22[1] := FALSE;
   STAT22[2] := FALSE;
   STAT22[3] := TRUE;
   STAT22[4] := FALSE;
   STAT22[5] := FALSE;
   STAT22[6] := FALSE;
   STAT22[7] := FALSE;
   STAT22[8] := TRUE;
   STAT22[9] := FALSE;
   STAT22[10] := FALSE;
   STAT22[11] := FALSE;
   STAT22[12] := FALSE;
   STAT22[13] := FALSE;
   STAT22[14] := FALSE;
   STAT22[15] := FALSE;
   STAT22[16] := FALSE;
   STAT22[17] := FALSE;
   STAT22[18] := FALSE;
   STAT22[19] := FALSE;
   STAT22[20] := FALSE;
   STAT22[21] := FALSE;
   STAT22[22] := FALSE;
   STAT22[23] := FALSE;
   STAT22[24] := FALSE;
   STAT22[25] := FALSE;
   STAT22[26] := FALSE;
   STAT22[27] := FALSE;
   STAT22[28] := FALSE;
   STAT22[29] := FALSE;
   STAT22[30] := FALSE;
   STAT22[31] := FALSE;
   STAT22[32] := FALSE;
   STAT22[33] := FALSE;
   STAT22[34] := FALSE;
   STAT22[35] := FALSE;
   STAT22[36] := FALSE;
   STAT22[37] := FALSE;
   STAT22[38] := FALSE;
   STAT22[39] := FALSE;
   STAT22[40] := FALSE;
   STAT23[1] := FALSE;
   STAT23[2] := TRUE;
   STAT23[3] := FALSE;
   STAT23[4] := FALSE;
   STAT23[5] := FALSE;
   STAT23[6] := TRUE;
   STAT23[7] := FALSE;
   STAT23[8] := FALSE;
   STAT23[9] := FALSE;
   STAT23[10] := FALSE;
   STAT23[11] := FALSE;
   STAT23[12] := FALSE;
   STAT23[13] := FALSE;
   STAT23[14] := FALSE;
   STAT23[15] := FALSE;
   STAT23[16] := FALSE;
   STAT23[17] := FALSE;
   STAT23[18] := FALSE;
   STAT23[19] := FALSE;
   STAT23[20] := FALSE;
   STAT23[21] := FALSE;
   STAT23[22] := FALSE;
   STAT23[23] := FALSE;
   STAT23[24] := FALSE;
   STAT23[25] := FALSE;
   STAT23[26] := FALSE;
   STAT23[27] := FALSE;
   STAT23[28] := FALSE;
   STAT23[29] := FALSE;
   STAT23[30] := FALSE;
   STAT23[31] := FALSE;
   STAT23[32] := FALSE;
   STAT23[33] := FALSE;
   STAT23[34] := FALSE;
   STAT23[35] := FALSE;
   STAT23[36] := FALSE;
   STAT23[37] := FALSE;
   STAT23[38] := FALSE;
   STAT23[39] := FALSE;
   STAT23[40] := FALSE;
   STAT24 := W#16#0;
   STAT25 := W#16#0;
   STAT26 := W#16#0;
   STAT27 := W#16#0;
   STAT28 := W#16#0;
   STAT29 := W#16#0;
   STAT30 := W#16#0;
   STAT31[1] := W#16#0;
   STAT31[2] := W#16#0;
   STAT31[3] := W#16#0;
   STAT31[4] := W#16#0;
   STAT31[5] := W#16#0;
   STAT31[6] := W#16#0;
   STAT31[7] := W#16#0;
   STAT32 := 100;
   STAT33 := 90;
   STAT34 := 80;
   STAT35 := 0;
   STAT36[1] := W#16#300;
   STAT36[2] := W#16#1418;
   STAT36[3] := W#16#3207;
   STAT36[4] := W#16#B;
   STAT36[5] := W#16#2716;
   STAT36[6] := W#16#200;
   STAT36[7] := W#16#1418;
   STAT36[8] := W#16#3205;
   STAT36[9] := W#16#1;
   STAT36[10] := W#16#2715;
   STAT36[11] := W#16#500;
   STAT36[12] := W#16#1418;
   STAT36[13] := W#16#3155;
   STAT36[14] := W#16#0;
   STAT36[15] := W#16#0;
   STAT36[16] := W#16#400;
   STAT36[17] := W#16#1418;
   STAT36[18] := W#16#2438;
   STAT36[19] := W#16#0;
   STAT36[20] := W#16#2715;
   STAT36[21] := W#16#300;
   STAT36[22] := W#16#1418;
   STAT36[23] := W#16#2347;
   STAT36[24] := W#16#B;
   STAT36[25] := W#16#2715;
   STAT36[26] := W#16#200;
   STAT36[27] := W#16#1418;
   STAT36[28] := W#16#2346;
   STAT36[29] := W#16#1;
   STAT36[30] := W#16#2714;
   STAT36[31] := W#16#500;
   STAT36[32] := W#16#1418;
   STAT36[33] := W#16#2337;
   STAT36[34] := W#16#0;
   STAT36[35] := W#16#0;
   STAT36[36] := W#16#400;
   STAT36[37] := W#16#1418;
   STAT36[38] := W#16#2324;
   STAT36[39] := W#16#0;
   STAT36[40] := W#16#2714;
   STAT36[41] := W#16#300;
   STAT36[42] := W#16#1418;
   STAT36[43] := W#16#2233;
   STAT36[44] := W#16#B;
   STAT36[45] := W#16#2714;
   STAT36[46] := W#16#200;
   STAT36[47] := W#16#1418;
   STAT36[48] := W#16#2231;
   STAT36[49] := W#16#1;
   STAT36[50] := W#16#2713;
   STAT36[51] := W#16#500;
   STAT36[52] := W#16#1418;
   STAT36[53] := W#16#2222;
   STAT36[54] := W#16#0;
   STAT36[55] := W#16#0;
   STAT36[56] := W#16#400;
   STAT36[57] := W#16#1418;
   STAT36[58] := W#16#2209;
   STAT36[59] := W#16#0;
   STAT36[60] := W#16#2713;
   STAT36[61] := W#16#300;
   STAT36[62] := W#16#1418;
   STAT36[63] := W#16#2117;
   STAT36[64] := W#16#B;
   STAT36[65] := W#16#2713;
   STAT36[66] := W#16#200;
   STAT36[67] := W#16#1418;
   STAT36[68] := W#16#2116;
   STAT36[69] := W#16#1;
   STAT36[70] := W#16#2712;
   STAT36[71] := W#16#500;
   STAT36[72] := W#16#1418;
   STAT36[73] := W#16#2107;
   STAT36[74] := W#16#0;
   STAT36[75] := W#16#0;
   STAT36[76] := W#16#400;
   STAT36[77] := W#16#1418;
   STAT36[78] := W#16#2054;
   STAT36[79] := W#16#0;
   STAT36[80] := W#16#2712;
   STAT36[81] := W#16#300;
   STAT36[82] := W#16#1418;
   STAT36[83] := W#16#2005;
   STAT36[84] := W#16#B;
   STAT36[85] := W#16#2712;
   STAT36[86] := W#16#200;
   STAT36[87] := W#16#1418;
   STAT36[88] := W#16#2004;
   STAT36[89] := W#16#1;
   STAT36[90] := W#16#2711;
   STAT36[91] := W#16#500;
   STAT36[92] := W#16#1418;
   STAT36[93] := W#16#1955;
   STAT36[94] := W#16#0;
   STAT36[95] := W#16#0;
   STAT36[96] := W#16#400;
   STAT36[97] := W#16#1418;
   STAT36[98] := W#16#1942;
   STAT36[99] := W#16#0;
   STAT36[100] := W#16#2711;
   STAT36[101] := W#16#300;
   STAT36[102] := W#16#1418;
   STAT36[103] := W#16#1851;
   STAT36[104] := W#16#B;
   STAT36[105] := W#16#2711;
   STAT36[106] := W#16#200;
   STAT36[107] := W#16#1418;
   STAT36[108] := W#16#1850;
   STAT36[109] := W#16#1;
   STAT36[110] := W#16#2710;
   STAT36[111] := W#16#500;
   STAT36[112] := W#16#1418;
   STAT36[113] := W#16#1842;
   STAT36[114] := W#16#0;
   STAT36[115] := W#16#0;
   STAT36[116] := W#16#400;
   STAT36[117] := W#16#1418;
   STAT36[118] := W#16#1828;
   STAT36[119] := W#16#0;
   STAT36[120] := W#16#2710;
   STAT36[121] := W#16#300;
   STAT36[122] := W#16#1418;
   STAT36[123] := W#16#1738;
   STAT36[124] := W#16#B;
   STAT36[125] := W#16#2710;
   STAT36[126] := W#16#200;
   STAT36[127] := W#16#1418;
   STAT36[128] := W#16#1737;
   STAT36[129] := W#16#1;
   STAT36[130] := W#16#2709;
   STAT36[131] := W#16#500;
   STAT36[132] := W#16#1418;
   STAT36[133] := W#16#1729;
   STAT36[134] := W#16#0;
   STAT36[135] := W#16#0;
   STAT36[136] := W#16#400;
   STAT36[137] := W#16#1418;
   STAT36[138] := W#16#1715;
   STAT36[139] := W#16#0;
   STAT36[140] := W#16#2709;
   STAT36[141] := W#16#300;
   STAT36[142] := W#16#1418;
   STAT36[143] := W#16#1627;
   STAT36[144] := W#16#B;
   STAT36[145] := W#16#2709;
   STAT36[146] := W#16#200;
   STAT36[147] := W#16#1418;
   STAT36[148] := W#16#1625;
   STAT36[149] := W#16#1;
   STAT36[150] := W#16#2708;
   STAT36[151] := W#16#500;
   STAT36[152] := W#16#1418;
   STAT36[153] := W#16#1615;
   STAT36[154] := W#16#0;
   STAT36[155] := W#16#0;
   STAT36[156] := W#16#400;
   STAT36[157] := W#16#1418;
   STAT36[158] := W#16#1603;
   STAT36[159] := W#16#0;
   STAT36[160] := W#16#2708;
   STAT36[161] := W#16#300;
   STAT36[162] := W#16#1418;
   STAT36[163] := W#16#1512;
   STAT36[164] := W#16#B;
   STAT36[165] := W#16#2708;
   STAT36[166] := W#16#200;
   STAT36[167] := W#16#1418;
   STAT36[168] := W#16#1511;
   STAT36[169] := W#16#1;
   STAT36[170] := W#16#2707;
   STAT36[171] := W#16#500;
   STAT36[172] := W#16#1418;
   STAT36[173] := W#16#1501;
   STAT36[174] := W#16#0;
   STAT36[175] := W#16#0;
   STAT36[176] := W#16#400;
   STAT36[177] := W#16#1418;
   STAT36[178] := W#16#1449;
   STAT36[179] := W#16#0;
   STAT36[180] := W#16#2707;
   STAT36[181] := W#16#300;
   STAT36[182] := W#16#1418;
   STAT36[183] := W#16#1359;
   STAT36[184] := W#16#B;
   STAT36[185] := W#16#2707;
   STAT36[186] := W#16#200;
   STAT36[187] := W#16#1418;
   STAT36[188] := W#16#1357;
   STAT36[189] := W#16#1;
   STAT36[190] := W#16#2706;
   STAT36[191] := W#16#500;
   STAT36[192] := W#16#1418;
   STAT36[193] := W#16#1347;
   STAT36[194] := W#16#0;
   STAT36[195] := W#16#0;
   STAT36[196] := W#16#400;
   STAT36[197] := W#16#1418;
   STAT36[198] := W#16#1335;
   STAT36[199] := W#16#0;
   STAT36[200] := W#16#2706;
   STAT36[201] := W#16#300;
   STAT36[202] := W#16#1418;
   STAT36[203] := W#16#1246;
   STAT36[204] := W#16#B;
   STAT36[205] := W#16#2706;
   STAT36[206] := W#16#200;
   STAT36[207] := W#16#1418;
   STAT36[208] := W#16#1245;
   STAT36[209] := W#16#1;
   STAT36[210] := W#16#2705;
   STAT36[211] := W#16#500;
   STAT36[212] := W#16#1418;
   STAT36[213] := W#16#1235;
   STAT36[214] := W#16#0;
   STAT36[215] := W#16#0;
   STAT36[216] := W#16#400;
   STAT36[217] := W#16#1418;
   STAT36[218] := W#16#1223;
   STAT36[219] := W#16#0;
   STAT36[220] := W#16#2705;
   STAT36[221] := W#16#300;
   STAT36[222] := W#16#1418;
   STAT36[223] := W#16#1132;
   STAT36[224] := W#16#B;
   STAT36[225] := W#16#2705;
   STAT36[226] := W#16#200;
   STAT36[227] := W#16#1418;
   STAT36[228] := W#16#1131;
   STAT36[229] := W#16#1;
   STAT36[230] := W#16#2704;
   STAT36[231] := W#16#500;
   STAT36[232] := W#16#1418;
   STAT36[233] := W#16#1121;
   STAT36[234] := W#16#0;
   STAT36[235] := W#16#0;
   STAT36[236] := W#16#400;
   STAT36[237] := W#16#1418;
   STAT36[238] := W#16#1109;
   STAT36[239] := W#16#0;
   STAT36[240] := W#16#2704;
   STAT36[241] := W#16#300;
   STAT36[242] := W#16#1418;
   STAT36[243] := W#16#1020;
   STAT36[244] := W#16#B;
   STAT36[245] := W#16#2704;
   STAT36[246] := W#16#200;
   STAT36[247] := W#16#1418;
   STAT36[248] := W#16#1019;
   STAT36[249] := W#16#1;
   STAT36[250] := W#16#2703;
   STAT36[251] := W#16#500;
   STAT36[252] := W#16#1418;
   STAT36[253] := W#16#1010;
   STAT36[254] := W#16#0;
   STAT36[255] := W#16#0;
   STAT36[256] := W#16#400;
   STAT36[257] := W#16#1418;
   STAT36[258] := W#16#957;
   STAT36[259] := W#16#0;
   STAT36[260] := W#16#2703;
   STAT36[261] := W#16#300;
   STAT36[262] := W#16#1418;
   STAT36[263] := W#16#904;
   STAT36[264] := W#16#B;
   STAT36[265] := W#16#2703;
   STAT36[266] := W#16#200;
   STAT36[267] := W#16#1418;
   STAT36[268] := W#16#903;
   STAT36[269] := W#16#1;
   STAT36[270] := W#16#2702;
   STAT36[271] := W#16#500;
   STAT36[272] := W#16#1418;
   STAT36[273] := W#16#854;
   STAT36[274] := W#16#0;
   STAT36[275] := W#16#0;
   STAT36[276] := W#16#400;
   STAT36[277] := W#16#1418;
   STAT36[278] := W#16#841;
   STAT36[279] := W#16#0;
   STAT36[280] := W#16#2702;
   STAT36[281] := W#16#300;
   STAT36[282] := W#16#1418;
   STAT36[283] := W#16#721;
   STAT36[284] := W#16#B;
   STAT36[285] := W#16#2702;
   STAT36[286] := W#16#200;
   STAT36[287] := W#16#1418;
   STAT36[288] := W#16#720;
   STAT36[289] := W#16#1;
   STAT36[290] := W#16#2701;
   STAT36[291] := W#16#500;
   STAT36[292] := W#16#1418;
   STAT36[293] := W#16#711;
   STAT36[294] := W#16#0;
   STAT36[295] := W#16#0;
   STAT36[296] := W#16#400;
   STAT36[297] := W#16#1418;
   STAT36[298] := W#16#658;
   STAT36[299] := W#16#0;
   STAT36[300] := W#16#2701;
   STAT36[301] := W#16#300;
   STAT36[302] := W#16#1418;
   STAT36[303] := W#16#343;
   STAT36[304] := W#16#B;
   STAT36[305] := W#16#2701;
   STAT36[306] := W#16#200;
   STAT36[307] := W#16#1418;
   STAT36[308] := W#16#342;
   STAT36[309] := W#16#1;
   STAT36[310] := W#16#2700;
   STAT36[311] := W#16#500;
   STAT36[312] := W#16#1418;
   STAT36[313] := W#16#333;
   STAT36[314] := W#16#0;
   STAT36[315] := W#16#0;
   STAT36[316] := W#16#400;
   STAT36[317] := W#16#1418;
   STAT36[318] := W#16#320;
   STAT36[319] := W#16#0;
   STAT36[320] := W#16#2700;
   STAT36[321] := W#16#300;
   STAT36[322] := W#16#1418;
   STAT36[323] := W#16#230;
   STAT36[324] := W#16#B;
   STAT36[325] := W#16#2700;
   STAT36[326] := W#16#200;
   STAT36[327] := W#16#1418;
   STAT36[328] := W#16#228;
   STAT36[329] := W#16#1;
   STAT36[330] := W#16#2699;
   STAT36[331] := W#16#500;
   STAT36[332] := W#16#1418;
   STAT36[333] := W#16#218;
   STAT36[334] := W#16#0;
   STAT36[335] := W#16#0;
   STAT36[336] := W#16#400;
   STAT36[337] := W#16#1418;
   STAT36[338] := W#16#206;
   STAT36[339] := W#16#0;
   STAT36[340] := W#16#2699;
   STAT36[341] := W#16#300;
   STAT36[342] := W#16#1418;
   STAT36[343] := W#16#112;
   STAT36[344] := W#16#B;
   STAT36[345] := W#16#2699;
   STAT36[346] := W#16#200;
   STAT36[347] := W#16#1418;
   STAT36[348] := W#16#111;
   STAT36[349] := W#16#1;
   STAT36[350] := W#16#2698;
   STAT36[351] := W#16#500;
   STAT36[352] := W#16#1418;
   STAT36[353] := W#16#101;
   STAT36[354] := W#16#0;
   STAT36[355] := W#16#0;
   STAT36[356] := W#16#400;
   STAT36[357] := W#16#1418;
   STAT36[358] := W#16#49;
   STAT36[359] := W#16#0;
   STAT36[360] := W#16#2698;
   STAT36[361] := W#16#300;
   STAT36[362] := W#16#1418;
   STAT36[363] := W#16#1;
   STAT36[364] := W#16#B;
   STAT36[365] := W#16#2698;
   STAT36[366] := W#16#200;
   STAT36[367] := W#16#1417;
   STAT36[368] := W#16#5959;
   STAT36[369] := W#16#1;
   STAT36[370] := W#16#2697;
   STAT36[371] := W#16#500;
   STAT36[372] := W#16#1417;
   STAT36[373] := W#16#5948;
   STAT36[374] := W#16#0;
   STAT36[375] := W#16#0;
   STAT36[376] := W#16#400;
   STAT36[377] := W#16#1417;
   STAT36[378] := W#16#5937;
   STAT36[379] := W#16#0;
   STAT36[380] := W#16#2697;
   STAT36[381] := W#16#300;
   STAT36[382] := W#16#1417;
   STAT36[383] := W#16#5845;
   STAT36[384] := W#16#B;
   STAT36[385] := W#16#2697;
   STAT36[386] := W#16#200;
   STAT36[387] := W#16#1417;
   STAT36[388] := W#16#5843;
   STAT36[389] := W#16#1;
   STAT36[390] := W#16#2696;
   STAT36[391] := W#16#500;
   STAT36[392] := W#16#1417;
   STAT36[393] := W#16#5834;
   STAT36[394] := W#16#0;
   STAT36[395] := W#16#0;
   STAT36[396] := W#16#400;
   STAT36[397] := W#16#1417;
   STAT36[398] := W#16#5821;
   STAT36[399] := W#16#0;
   STAT36[400] := W#16#2696;
   STAT36[401] := W#16#300;
   STAT36[402] := W#16#1417;
   STAT36[403] := W#16#5730;
   STAT36[404] := W#16#B;
   STAT36[405] := W#16#2696;
   STAT36[406] := W#16#200;
   STAT36[407] := W#16#1417;
   STAT36[408] := W#16#5728;
   STAT36[409] := W#16#1;
   STAT36[410] := W#16#2695;
   STAT36[411] := W#16#500;
   STAT36[412] := W#16#1417;
   STAT36[413] := W#16#5719;
   STAT36[414] := W#16#0;
   STAT36[415] := W#16#0;
   STAT36[416] := W#16#400;
   STAT36[417] := W#16#1417;
   STAT36[418] := W#16#5706;
   STAT36[419] := W#16#0;
   STAT36[420] := W#16#2695;
   STAT36[421] := W#16#300;
   STAT36[422] := W#16#1417;
   STAT36[423] := W#16#5617;
   STAT36[424] := W#16#B;
   STAT36[425] := W#16#2695;
   STAT36[426] := W#16#200;
   STAT36[427] := W#16#1417;
   STAT36[428] := W#16#5616;
   STAT36[429] := W#16#1;
   STAT36[430] := W#16#2694;
   STAT36[431] := W#16#500;
   STAT36[432] := W#16#1417;
   STAT36[433] := W#16#5607;
   STAT36[434] := W#16#0;
   STAT36[435] := W#16#0;
   STAT36[436] := W#16#400;
   STAT36[437] := W#16#1417;
   STAT36[438] := W#16#5554;
   STAT36[439] := W#16#0;
   STAT36[440] := W#16#2694;
   STAT36[441] := W#16#300;
   STAT36[442] := W#16#1417;
   STAT36[443] := W#16#5504;
   STAT36[444] := W#16#B;
   STAT36[445] := W#16#2694;
   STAT36[446] := W#16#200;
   STAT36[447] := W#16#1417;
   STAT36[448] := W#16#5503;
   STAT36[449] := W#16#1;
   STAT36[450] := W#16#2693;
   STAT36[451] := W#16#500;
   STAT36[452] := W#16#1417;
   STAT36[453] := W#16#5454;
   STAT36[454] := W#16#0;
   STAT36[455] := W#16#0;
   STAT36[456] := W#16#400;
   STAT36[457] := W#16#1417;
   STAT36[458] := W#16#5441;
   STAT36[459] := W#16#0;
   STAT36[460] := W#16#2693;
   STAT36[461] := W#16#300;
   STAT36[462] := W#16#1417;
   STAT36[463] := W#16#5351;
   STAT36[464] := W#16#B;
   STAT36[465] := W#16#2693;
   STAT36[466] := W#16#200;
   STAT36[467] := W#16#1417;
   STAT36[468] := W#16#5350;
   STAT36[469] := W#16#1;
   STAT36[470] := W#16#2692;
   STAT36[471] := W#16#500;
   STAT36[472] := W#16#1417;
   STAT36[473] := W#16#5341;
   STAT36[474] := W#16#0;
   STAT36[475] := W#16#0;
   STAT36[476] := W#16#400;
   STAT36[477] := W#16#1417;
   STAT36[478] := W#16#5328;
   STAT36[479] := W#16#0;
   STAT36[480] := W#16#2692;
   STAT36[481] := W#16#300;
   STAT36[482] := W#16#1417;
   STAT36[483] := W#16#5237;
   STAT36[484] := W#16#B;
   STAT36[485] := W#16#2692;
   STAT36[486] := W#16#200;
   STAT36[487] := W#16#1417;
   STAT36[488] := W#16#5236;
   STAT36[489] := W#16#1;
   STAT36[490] := W#16#2691;
   STAT36[491] := W#16#500;
   STAT36[492] := W#16#1417;
   STAT36[493] := W#16#5227;
   STAT36[494] := W#16#0;
   STAT36[495] := W#16#0;
   STAT36[496] := W#16#400;
   STAT36[497] := W#16#1417;
   STAT36[498] := W#16#5214;
   STAT36[499] := W#16#0;
   STAT36[500] := W#16#2691;
   STAT37[1] := B#16#0;
   STAT37[2] := B#16#87;
   STAT37[3] := B#16#27;
   STAT37[4] := B#16#16;
   STAT37[5] := B#16#22;
   STAT37[6] := B#16#22;
   STAT37[7] := B#16#80;
   STAT37[8] := B#16#4;
   STAT37[9] := B#16#16;
   STAT37[10] := B#16#10;
   STAT37[11] := B#16#60;
   STAT37[12] := B#16#0;
   STAT37[13] := B#16#0;
   STAT37[14] := B#16#0;
   STAT37[15] := B#16#0;
   STAT37[16] := B#16#0;
   STAT38[1] := B#16#0;
   STAT38[2] := B#16#0;
   STAT38[3] := B#16#0;
   STAT38[4] := B#16#0;
   STAT39[1] := B#16#27;
   STAT39[2] := B#16#16;
   STAT39[3] := B#16#0;
   STAT39[4] := B#16#87;
   STAT39[5] := B#16#22;
   STAT39[6] := B#16#22;
   STAT39[7] := B#16#4;
   STAT39[8] := B#16#80;
   STAT39[9] := B#16#10;
   STAT39[10] := B#16#16;
   STAT39[11] := B#16#0;
   STAT39[12] := B#16#60;
   STAT39[13] := B#16#0;
   STAT39[14] := B#16#0;
   STAT39[15] := B#16#0;
   STAT39[16] := B#16#0;
END_DATA_BLOCK

DATA_BLOCK DB 166
VERSION : 0.1


  STRUCT
   STAT0 : WORD ;
   STAT1 : WORD ;
   STAT2 : WORD ;
   STAT3 : WORD ;
   STAT4 : WORD ;
   STAT5 : WORD ;
   STAT6 : WORD ;
   STAT7 : WORD ;
   STAT8 : WORD ;
   STAT9 : WORD ;
   STAT10 : WORD ;
   STAT11 : WORD ;
   STAT12 : WORD ;
   STAT13 : WORD ;
   STAT14 : WORD ;
   STAT15 : WORD ;
   STAT16 : INT ;
   STAT17 : INT ;
   STAT18 : INT ;
   STAT19 : INT ;
   STAT20 : ARRAY  [1 .. 6 ] OF BYTE ;
   STAT21 : ARRAY  [1 .. 6 ] OF BYTE ;
   STAT22 : ARRAY  [1 .. 40 ] OF BOOL  := FALSE;
   STAT23 : ARRAY  [1 .. 40 ] OF BOOL  := FALSE;
   STAT24 : WORD ;
   STAT25 : WORD ;
   STAT26 : WORD ;
   STAT27 : WORD ;
   STAT28 : WORD ;
   STAT29 : WORD ;
   STAT30 : WORD ;
   STAT31 : ARRAY  [1 .. 7 ] OF WORD ;
   STAT32 : INT ;
   STAT33 : INT ;
   STAT34 : INT ;
   STAT35 : INT ;
   STAT36 : ARRAY  [1 .. 500 ] OF WORD ;
   STAT37 : ARRAY  [1 .. 16 ] OF BYTE ;
   STAT38 : ARRAY  [1 .. 4 ] OF BYTE ;
   STAT39 : ARRAY  [1 .. 16 ] OF BYTE ;
  END_STRUCT ;
BEGIN
   STAT0 := W#16#2714;
   STAT1 := W#16#87;
   STAT2 := W#16#2222;
   STAT3 := W#16#180;
   STAT4 := W#16#5416;
   STAT5 := W#16#60;
   STAT6 := W#16#0;
   STAT7 := W#16#0;
   STAT8 := W#16#87;
   STAT9 := W#16#2714;
   STAT10 := W#16#2222;
   STAT11 := W#16#8001;
   STAT12 := W#16#1654;
   STAT13 := W#16#6000;
   STAT14 := W#16#0;
   STAT15 := W#16#0;
   STAT16 := 0;
   STAT17 := 3;
   STAT18 := 3;
   STAT19 := 0;
   STAT20[1] := B#16#0;
   STAT20[2] := B#16#0;
   STAT20[3] := B#16#0;
   STAT20[4] := B#16#0;
   STAT20[5] := B#16#0;
   STAT20[6] := B#16#0;
   STAT21[1] := B#16#0;
   STAT21[2] := B#16#0;
   STAT21[3] := B#16#0;
   STAT21[4] := B#16#0;
   STAT21[5] := B#16#0;
   STAT21[6] := B#16#0;
   STAT22[1] := FALSE;
   STAT22[2] := FALSE;
   STAT22[3] := TRUE;
   STAT22[4] := FALSE;
   STAT22[5] := FALSE;
   STAT22[6] := FALSE;
   STAT22[7] := FALSE;
   STAT22[8] := TRUE;
   STAT22[9] := FALSE;
   STAT22[10] := FALSE;
   STAT22[11] := FALSE;
   STAT22[12] := FALSE;
   STAT22[13] := FALSE;
   STAT22[14] := FALSE;
   STAT22[15] := FALSE;
   STAT22[16] := FALSE;
   STAT22[17] := FALSE;
   STAT22[18] := FALSE;
   STAT22[19] := FALSE;
   STAT22[20] := FALSE;
   STAT22[21] := FALSE;
   STAT22[22] := FALSE;
   STAT22[23] := FALSE;
   STAT22[24] := FALSE;
   STAT22[25] := FALSE;
   STAT22[26] := FALSE;
   STAT22[27] := FALSE;
   STAT22[28] := FALSE;
   STAT22[29] := FALSE;
   STAT22[30] := FALSE;
   STAT22[31] := FALSE;
   STAT22[32] := FALSE;
   STAT22[33] := FALSE;
   STAT22[34] := FALSE;
   STAT22[35] := FALSE;
   STAT22[36] := FALSE;
   STAT22[37] := FALSE;
   STAT22[38] := FALSE;
   STAT22[39] := FALSE;
   STAT22[40] := FALSE;
   STAT23[1] := FALSE;
   STAT23[2] := FALSE;
   STAT23[3] := TRUE;
   STAT23[4] := TRUE;
   STAT23[5] := TRUE;
   STAT23[6] := FALSE;
   STAT23[7] := FALSE;
   STAT23[8] := FALSE;
   STAT23[9] := FALSE;
   STAT23[10] := FALSE;
   STAT23[11] := FALSE;
   STAT23[12] := FALSE;
   STAT23[13] := FALSE;
   STAT23[14] := FALSE;
   STAT23[15] := FALSE;
   STAT23[16] := FALSE;
   STAT23[17] := FALSE;
   STAT23[18] := FALSE;
   STAT23[19] := FALSE;
   STAT23[20] := FALSE;
   STAT23[21] := FALSE;
   STAT23[22] := FALSE;
   STAT23[23] := FALSE;
   STAT23[24] := FALSE;
   STAT23[25] := FALSE;
   STAT23[26] := TRUE;
   STAT23[27] := FALSE;
   STAT23[28] := FALSE;
   STAT23[29] := FALSE;
   STAT23[30] := FALSE;
   STAT23[31] := FALSE;
   STAT23[32] := FALSE;
   STAT23[33] := FALSE;
   STAT23[34] := FALSE;
   STAT23[35] := FALSE;
   STAT23[36] := FALSE;
   STAT23[37] := FALSE;
   STAT23[38] := FALSE;
   STAT23[39] := FALSE;
   STAT23[40] := FALSE;
   STAT24 := W#16#400;
   STAT25 := W#16#400;
   STAT26 := W#16#0;
   STAT27 := W#16#0;
   STAT28 := W#16#0;
   STAT29 := W#16#0;
   STAT30 := W#16#0;
   STAT31[1] := W#16#0;
   STAT31[2] := W#16#0;
   STAT31[3] := W#16#0;
   STAT31[4] := W#16#0;
   STAT31[5] := W#16#0;
   STAT31[6] := W#16#0;
   STAT31[7] := W#16#0;
   STAT32 := 100;
   STAT33 := 90;
   STAT34 := 80;
   STAT35 := 0;
   STAT36[1] := W#16#400;
   STAT36[2] := W#16#1418;
   STAT36[3] := W#16#3257;
   STAT36[4] := W#16#0;
   STAT36[5] := W#16#2714;
   STAT36[6] := W#16#300;
   STAT36[7] := W#16#1418;
   STAT36[8] := W#16#3240;
   STAT36[9] := W#16#B;
   STAT36[10] := W#16#2714;
   STAT36[11] := W#16#200;
   STAT36[12] := W#16#1418;
   STAT36[13] := W#16#3238;
   STAT36[14] := W#16#1;
   STAT36[15] := W#16#4602;
   STAT36[16] := W#16#500;
   STAT36[17] := W#16#1418;
   STAT36[18] := W#16#3238;
   STAT36[19] := W#16#0;
   STAT36[20] := W#16#2714;
   STAT36[21] := W#16#400;
   STAT36[22] := W#16#1418;
   STAT36[23] := W#16#3228;
   STAT36[24] := W#16#0;
   STAT36[25] := W#16#2713;
   STAT36[26] := W#16#300;
   STAT36[27] := W#16#1418;
   STAT36[28] := W#16#3125;
   STAT36[29] := W#16#B;
   STAT36[30] := W#16#2713;
   STAT36[31] := W#16#200;
   STAT36[32] := W#16#1418;
   STAT36[33] := W#16#3124;
   STAT36[34] := W#16#1;
   STAT36[35] := W#16#4602;
   STAT36[36] := W#16#500;
   STAT36[37] := W#16#1418;
   STAT36[38] := W#16#3124;
   STAT36[39] := W#16#0;
   STAT36[40] := W#16#2713;
   STAT36[41] := W#16#400;
   STAT36[42] := W#16#1418;
   STAT36[43] := W#16#2248;
   STAT36[44] := W#16#0;
   STAT36[45] := W#16#2712;
   STAT36[46] := W#16#300;
   STAT36[47] := W#16#1418;
   STAT36[48] := W#16#2231;
   STAT36[49] := W#16#B;
   STAT36[50] := W#16#2712;
   STAT36[51] := W#16#200;
   STAT36[52] := W#16#1418;
   STAT36[53] := W#16#2229;
   STAT36[54] := W#16#1;
   STAT36[55] := W#16#4602;
   STAT36[56] := W#16#500;
   STAT36[57] := W#16#1418;
   STAT36[58] := W#16#2229;
   STAT36[59] := W#16#0;
   STAT36[60] := W#16#2712;
   STAT36[61] := W#16#400;
   STAT36[62] := W#16#1418;
   STAT36[63] := W#16#2211;
   STAT36[64] := W#16#0;
   STAT36[65] := W#16#2711;
   STAT36[66] := W#16#300;
   STAT36[67] := W#16#1418;
   STAT36[68] := W#16#2120;
   STAT36[69] := W#16#B;
   STAT36[70] := W#16#2711;
   STAT36[71] := W#16#200;
   STAT36[72] := W#16#1418;
   STAT36[73] := W#16#2119;
   STAT36[74] := W#16#1;
   STAT36[75] := W#16#4602;
   STAT36[76] := W#16#500;
   STAT36[77] := W#16#1418;
   STAT36[78] := W#16#2119;
   STAT36[79] := W#16#0;
   STAT36[80] := W#16#2711;
   STAT36[81] := W#16#400;
   STAT36[82] := W#16#1418;
   STAT36[83] := W#16#2044;
   STAT36[84] := W#16#0;
   STAT36[85] := W#16#2710;
   STAT36[86] := W#16#300;
   STAT36[87] := W#16#1418;
   STAT36[88] := W#16#2004;
   STAT36[89] := W#16#B;
   STAT36[90] := W#16#2710;
   STAT36[91] := W#16#200;
   STAT36[92] := W#16#1418;
   STAT36[93] := W#16#2003;
   STAT36[94] := W#16#1;
   STAT36[95] := W#16#4602;
   STAT36[96] := W#16#500;
   STAT36[97] := W#16#1418;
   STAT36[98] := W#16#2003;
   STAT36[99] := W#16#0;
   STAT36[100] := W#16#2710;
   STAT36[101] := W#16#400;
   STAT36[102] := W#16#1418;
   STAT36[103] := W#16#1921;
   STAT36[104] := W#16#0;
   STAT36[105] := W#16#2709;
   STAT36[106] := W#16#300;
   STAT36[107] := W#16#1418;
   STAT36[108] := W#16#1851;
   STAT36[109] := W#16#B;
   STAT36[110] := W#16#2709;
   STAT36[111] := W#16#200;
   STAT36[112] := W#16#1418;
   STAT36[113] := W#16#1850;
   STAT36[114] := W#16#1;
   STAT36[115] := W#16#4602;
   STAT36[116] := W#16#500;
   STAT36[117] := W#16#1418;
   STAT36[118] := W#16#1850;
   STAT36[119] := W#16#0;
   STAT36[120] := W#16#2709;
   STAT36[121] := W#16#400;
   STAT36[122] := W#16#1418;
   STAT36[123] := W#16#1757;
   STAT36[124] := W#16#0;
   STAT36[125] := W#16#2708;
   STAT36[126] := W#16#300;
   STAT36[127] := W#16#1418;
   STAT36[128] := W#16#1740;
   STAT36[129] := W#16#B;
   STAT36[130] := W#16#2708;
   STAT36[131] := W#16#200;
   STAT36[132] := W#16#1418;
   STAT36[133] := W#16#1739;
   STAT36[134] := W#16#1;
   STAT36[135] := W#16#4602;
   STAT36[136] := W#16#500;
   STAT36[137] := W#16#1418;
   STAT36[138] := W#16#1739;
   STAT36[139] := W#16#0;
   STAT36[140] := W#16#2708;
   STAT36[141] := W#16#400;
   STAT36[142] := W#16#1418;
   STAT36[143] := W#16#1643;
   STAT36[144] := W#16#0;
   STAT36[145] := W#16#2707;
   STAT36[146] := W#16#300;
   STAT36[147] := W#16#1418;
   STAT36[148] := W#16#1625;
   STAT36[149] := W#16#B;
   STAT36[150] := W#16#2707;
   STAT36[151] := W#16#200;
   STAT36[152] := W#16#1418;
   STAT36[153] := W#16#1623;
   STAT36[154] := W#16#1;
   STAT36[155] := W#16#4602;
   STAT36[156] := W#16#500;
   STAT36[157] := W#16#1418;
   STAT36[158] := W#16#1623;
   STAT36[159] := W#16#0;
   STAT36[160] := W#16#2707;
   STAT36[161] := W#16#400;
   STAT36[162] := W#16#1418;
   STAT36[163] := W#16#1541;
   STAT36[164] := W#16#0;
   STAT36[165] := W#16#2706;
   STAT36[166] := W#16#300;
   STAT36[167] := W#16#1418;
   STAT36[168] := W#16#1511;
   STAT36[169] := W#16#B;
   STAT36[170] := W#16#2706;
   STAT36[171] := W#16#200;
   STAT36[172] := W#16#1418;
   STAT36[173] := W#16#1510;
   STAT36[174] := W#16#1;
   STAT36[175] := W#16#4602;
   STAT36[176] := W#16#500;
   STAT36[177] := W#16#1418;
   STAT36[178] := W#16#1510;
   STAT36[179] := W#16#0;
   STAT36[180] := W#16#2706;
   STAT36[181] := W#16#400;
   STAT36[182] := W#16#1418;
   STAT36[183] := W#16#1430;
   STAT36[184] := W#16#0;
   STAT36[185] := W#16#2705;
   STAT36[186] := W#16#300;
   STAT36[187] := W#16#1418;
   STAT36[188] := W#16#1401;
   STAT36[189] := W#16#B;
   STAT36[190] := W#16#2705;
   STAT36[191] := W#16#200;
   STAT36[192] := W#16#1418;
   STAT36[193] := W#16#1359;
   STAT36[194] := W#16#1;
   STAT36[195] := W#16#4602;
   STAT36[196] := W#16#500;
   STAT36[197] := W#16#1418;
   STAT36[198] := W#16#1359;
   STAT36[199] := W#16#0;
   STAT36[200] := W#16#2705;
   STAT36[201] := W#16#400;
   STAT36[202] := W#16#1418;
   STAT36[203] := W#16#1318;
   STAT36[204] := W#16#0;
   STAT36[205] := W#16#2704;
   STAT36[206] := W#16#300;
   STAT36[207] := W#16#1418;
   STAT36[208] := W#16#1245;
   STAT36[209] := W#16#B;
   STAT36[210] := W#16#2704;
   STAT36[211] := W#16#200;
   STAT36[212] := W#16#1418;
   STAT36[213] := W#16#1244;
   STAT36[214] := W#16#1;
   STAT36[215] := W#16#4602;
   STAT36[216] := W#16#500;
   STAT36[217] := W#16#1418;
   STAT36[218] := W#16#1244;
   STAT36[219] := W#16#0;
   STAT36[220] := W#16#2704;
   STAT36[221] := W#16#400;
   STAT36[222] := W#16#1418;
   STAT36[223] := W#16#1201;
   STAT36[224] := W#16#0;
   STAT36[225] := W#16#2703;
   STAT36[226] := W#16#300;
   STAT36[227] := W#16#1418;
   STAT36[228] := W#16#1130;
   STAT36[229] := W#16#B;
   STAT36[230] := W#16#2703;
   STAT36[231] := W#16#200;
   STAT36[232] := W#16#1418;
   STAT36[233] := W#16#1128;
   STAT36[234] := W#16#1;
   STAT36[235] := W#16#4602;
   STAT36[236] := W#16#500;
   STAT36[237] := W#16#1418;
   STAT36[238] := W#16#1128;
   STAT36[239] := W#16#0;
   STAT36[240] := W#16#2703;
   STAT36[241] := W#16#400;
   STAT36[242] := W#16#1418;
   STAT36[243] := W#16#1033;
   STAT36[244] := W#16#0;
   STAT36[245] := W#16#2702;
   STAT36[246] := W#16#300;
   STAT36[247] := W#16#1418;
   STAT36[248] := W#16#1014;
   STAT36[249] := W#16#B;
   STAT36[250] := W#16#2702;
   STAT36[251] := W#16#200;
   STAT36[252] := W#16#1418;
   STAT36[253] := W#16#1012;
   STAT36[254] := W#16#1;
   STAT36[255] := W#16#4602;
   STAT36[256] := W#16#500;
   STAT36[257] := W#16#1418;
   STAT36[258] := W#16#1012;
   STAT36[259] := W#16#0;
   STAT36[260] := W#16#2702;
   STAT36[261] := W#16#400;
   STAT36[262] := W#16#1418;
   STAT36[263] := W#16#925;
   STAT36[264] := W#16#0;
   STAT36[265] := W#16#2701;
   STAT36[266] := W#16#300;
   STAT36[267] := W#16#1418;
   STAT36[268] := W#16#858;
   STAT36[269] := W#16#B;
   STAT36[270] := W#16#2701;
   STAT36[271] := W#16#200;
   STAT36[272] := W#16#1418;
   STAT36[273] := W#16#857;
   STAT36[274] := W#16#1;
   STAT36[275] := W#16#4602;
   STAT36[276] := W#16#500;
   STAT36[277] := W#16#1418;
   STAT36[278] := W#16#857;
   STAT36[279] := W#16#0;
   STAT36[280] := W#16#2701;
   STAT36[281] := W#16#400;
   STAT36[282] := W#16#1418;
   STAT36[283] := W#16#834;
   STAT36[284] := W#16#0;
   STAT36[285] := W#16#2700;
   STAT36[286] := W#16#300;
   STAT36[287] := W#16#1418;
   STAT36[288] := W#16#746;
   STAT36[289] := W#16#B;
   STAT36[290] := W#16#2700;
   STAT36[291] := W#16#200;
   STAT36[292] := W#16#1418;
   STAT36[293] := W#16#744;
   STAT36[294] := W#16#1;
   STAT36[295] := W#16#4602;
   STAT36[296] := W#16#500;
   STAT36[297] := W#16#1418;
   STAT36[298] := W#16#744;
   STAT36[299] := W#16#0;
   STAT36[300] := W#16#2700;
   STAT36[301] := W#16#400;
   STAT36[302] := W#16#1418;
   STAT36[303] := W#16#659;
   STAT36[304] := W#16#0;
   STAT36[305] := W#16#2699;
   STAT36[306] := W#16#300;
   STAT36[307] := W#16#1418;
   STAT36[308] := W#16#632;
   STAT36[309] := W#16#B;
   STAT36[310] := W#16#2699;
   STAT36[311] := W#16#200;
   STAT36[312] := W#16#1418;
   STAT36[313] := W#16#630;
   STAT36[314] := W#16#1;
   STAT36[315] := W#16#4602;
   STAT36[316] := W#16#500;
   STAT36[317] := W#16#1418;
   STAT36[318] := W#16#630;
   STAT36[319] := W#16#0;
   STAT36[320] := W#16#2699;
   STAT36[321] := W#16#400;
   STAT36[322] := W#16#1418;
   STAT36[323] := W#16#257;
   STAT36[324] := W#16#0;
   STAT36[325] := W#16#2698;
   STAT36[326] := W#16#300;
   STAT36[327] := W#16#1418;
   STAT36[328] := W#16#226;
   STAT36[329] := W#16#B;
   STAT36[330] := W#16#2698;
   STAT36[331] := W#16#200;
   STAT36[332] := W#16#1418;
   STAT36[333] := W#16#224;
   STAT36[334] := W#16#1;
   STAT36[335] := W#16#4602;
   STAT36[336] := W#16#500;
   STAT36[337] := W#16#1418;
   STAT36[338] := W#16#224;
   STAT36[339] := W#16#0;
   STAT36[340] := W#16#2698;
   STAT36[341] := W#16#400;
   STAT36[342] := W#16#1418;
   STAT36[343] := W#16#156;
   STAT36[344] := W#16#0;
   STAT36[345] := W#16#2697;
   STAT36[346] := W#16#300;
   STAT36[347] := W#16#1418;
   STAT36[348] := W#16#112;
   STAT36[349] := W#16#B;
   STAT36[350] := W#16#2697;
   STAT36[351] := W#16#200;
   STAT36[352] := W#16#1418;
   STAT36[353] := W#16#111;
   STAT36[354] := W#16#1;
   STAT36[355] := W#16#4602;
   STAT36[356] := W#16#500;
   STAT36[357] := W#16#1418;
   STAT36[358] := W#16#111;
   STAT36[359] := W#16#0;
   STAT36[360] := W#16#2697;
   STAT36[361] := W#16#400;
   STAT36[362] := W#16#1418;
   STAT36[363] := W#16#21;
   STAT36[364] := W#16#0;
   STAT36[365] := W#16#2696;
   STAT36[366] := W#16#300;
   STAT36[367] := W#16#1417;
   STAT36[368] := W#16#5957;
   STAT36[369] := W#16#B;
   STAT36[370] := W#16#2696;
   STAT36[371] := W#16#200;
   STAT36[372] := W#16#1417;
   STAT36[373] := W#16#5955;
   STAT36[374] := W#16#1;
   STAT36[375] := W#16#4602;
   STAT36[376] := W#16#500;
   STAT36[377] := W#16#1417;
   STAT36[378] := W#16#5955;
   STAT36[379] := W#16#0;
   STAT36[380] := W#16#2696;
   STAT36[381] := W#16#400;
   STAT36[382] := W#16#1417;
   STAT36[383] := W#16#5932;
   STAT36[384] := W#16#0;
   STAT36[385] := W#16#2695;
   STAT36[386] := W#16#300;
   STAT36[387] := W#16#1417;
   STAT36[388] := W#16#5842;
   STAT36[389] := W#16#B;
   STAT36[390] := W#16#2695;
   STAT36[391] := W#16#200;
   STAT36[392] := W#16#1417;
   STAT36[393] := W#16#5840;
   STAT36[394] := W#16#1;
   STAT36[395] := W#16#4602;
   STAT36[396] := W#16#500;
   STAT36[397] := W#16#1417;
   STAT36[398] := W#16#5840;
   STAT36[399] := W#16#0;
   STAT36[400] := W#16#2695;
   STAT36[401] := W#16#400;
   STAT36[402] := W#16#1417;
   STAT36[403] := W#16#5749;
   STAT36[404] := W#16#0;
   STAT36[405] := W#16#2694;
   STAT36[406] := W#16#300;
   STAT36[407] := W#16#1417;
   STAT36[408] := W#16#5730;
   STAT36[409] := W#16#B;
   STAT36[410] := W#16#2694;
   STAT36[411] := W#16#200;
   STAT36[412] := W#16#1417;
   STAT36[413] := W#16#5729;
   STAT36[414] := W#16#1;
   STAT36[415] := W#16#4602;
   STAT36[416] := W#16#500;
   STAT36[417] := W#16#1417;
   STAT36[418] := W#16#5729;
   STAT36[419] := W#16#0;
   STAT36[420] := W#16#2694;
   STAT36[421] := W#16#400;
   STAT36[422] := W#16#1417;
   STAT36[423] := W#16#5648;
   STAT36[424] := W#16#0;
   STAT36[425] := W#16#2693;
   STAT36[426] := W#16#300;
   STAT36[427] := W#16#1417;
   STAT36[428] := W#16#5617;
   STAT36[429] := W#16#B;
   STAT36[430] := W#16#2693;
   STAT36[431] := W#16#200;
   STAT36[432] := W#16#1417;
   STAT36[433] := W#16#5616;
   STAT36[434] := W#16#1;
   STAT36[435] := W#16#4602;
   STAT36[436] := W#16#500;
   STAT36[437] := W#16#1417;
   STAT36[438] := W#16#5616;
   STAT36[439] := W#16#0;
   STAT36[440] := W#16#2693;
   STAT36[441] := W#16#400;
   STAT36[442] := W#16#1417;
   STAT36[443] := W#16#5534;
   STAT36[444] := W#16#0;
   STAT36[445] := W#16#2692;
   STAT36[446] := W#16#300;
   STAT36[447] := W#16#1417;
   STAT36[448] := W#16#5504;
   STAT36[449] := W#16#B;
   STAT36[450] := W#16#2692;
   STAT36[451] := W#16#200;
   STAT36[452] := W#16#1417;
   STAT36[453] := W#16#5503;
   STAT36[454] := W#16#1;
   STAT36[455] := W#16#4602;
   STAT36[456] := W#16#500;
   STAT36[457] := W#16#1417;
   STAT36[458] := W#16#5503;
   STAT36[459] := W#16#0;
   STAT36[460] := W#16#2692;
   STAT36[461] := W#16#400;
   STAT36[462] := W#16#1417;
   STAT36[463] := W#16#5423;
   STAT36[464] := W#16#0;
   STAT36[465] := W#16#2691;
   STAT36[466] := W#16#300;
   STAT36[467] := W#16#1417;
   STAT36[468] := W#16#5351;
   STAT36[469] := W#16#B;
   STAT36[470] := W#16#2691;
   STAT36[471] := W#16#200;
   STAT36[472] := W#16#1417;
   STAT36[473] := W#16#5349;
   STAT36[474] := W#16#1;
   STAT36[475] := W#16#4602;
   STAT36[476] := W#16#500;
   STAT36[477] := W#16#1417;
   STAT36[478] := W#16#5349;
   STAT36[479] := W#16#0;
   STAT36[480] := W#16#2691;
   STAT36[481] := W#16#400;
   STAT36[482] := W#16#1417;
   STAT36[483] := W#16#5305;
   STAT36[484] := W#16#0;
   STAT36[485] := W#16#2690;
   STAT36[486] := W#16#300;
   STAT36[487] := W#16#1417;
   STAT36[488] := W#16#5235;
   STAT36[489] := W#16#B;
   STAT36[490] := W#16#2690;
   STAT36[491] := W#16#200;
   STAT36[492] := W#16#1417;
   STAT36[493] := W#16#5234;
   STAT36[494] := W#16#1;
   STAT36[495] := W#16#4602;
   STAT36[496] := W#16#500;
   STAT36[497] := W#16#1417;
   STAT36[498] := W#16#5234;
   STAT36[499] := W#16#0;
   STAT36[500] := W#16#2690;
   STAT37[1] := B#16#0;
   STAT37[2] := B#16#87;
   STAT37[3] := B#16#27;
   STAT37[4] := B#16#14;
   STAT37[5] := B#16#22;
   STAT37[6] := B#16#22;
   STAT37[7] := B#16#80;
   STAT37[8] := B#16#1;
   STAT37[9] := B#16#16;
   STAT37[10] := B#16#54;
   STAT37[11] := B#16#60;
   STAT37[12] := B#16#0;
   STAT37[13] := B#16#0;
   STAT37[14] := B#16#0;
   STAT37[15] := B#16#0;
   STAT37[16] := B#16#0;
   STAT38[1] := B#16#0;
   STAT38[2] := B#16#0;
   STAT38[3] := B#16#0;
   STAT38[4] := B#16#0;
   STAT39[1] := B#16#27;
   STAT39[2] := B#16#14;
   STAT39[3] := B#16#0;
   STAT39[4] := B#16#87;
   STAT39[5] := B#16#22;
   STAT39[6] := B#16#22;
   STAT39[7] := B#16#1;
   STAT39[8] := B#16#80;
   STAT39[9] := B#16#54;
   STAT39[10] := B#16#16;
   STAT39[11] := B#16#0;
   STAT39[12] := B#16#60;
   STAT39[13] := B#16#0;
   STAT39[14] := B#16#0;
   STAT39[15] := B#16#0;
   STAT39[16] := B#16#0;
END_DATA_BLOCK

DATA_BLOCK DB 167
VERSION : 0.1


  STRUCT
   STAT0 : WORD ;
   STAT1 : WORD ;
   STAT2 : WORD ;
   STAT3 : WORD ;
   STAT4 : WORD ;
   STAT5 : WORD ;
   STAT6 : WORD ;
   STAT7 : WORD ;
   STAT8 : WORD ;
   STAT9 : WORD ;
   STAT10 : WORD ;
   STAT11 : WORD ;
   STAT12 : WORD ;
   STAT13 : WORD ;
   STAT14 : WORD ;
   STAT15 : WORD ;
   STAT16 : INT ;
   STAT17 : INT ;
   STAT18 : INT ;
   STAT19 : INT ;
   STAT20 : ARRAY  [1 .. 6 ] OF BYTE ;
   STAT21 : ARRAY  [1 .. 6 ] OF BYTE ;
   STAT22 : ARRAY  [1 .. 40 ] OF BOOL  := FALSE;
   STAT23 : ARRAY  [1 .. 40 ] OF BOOL  := FALSE;
   STAT24 : WORD ;
   STAT25 : WORD ;
   STAT26 : WORD ;
   STAT27 : WORD ;
   STAT28 : WORD ;
   STAT29 : WORD ;
   STAT30 : WORD ;
   STAT31 : ARRAY  [1 .. 7 ] OF WORD ;
   STAT32 : INT ;
   STAT33 : INT ;
   STAT34 : INT ;
   STAT35 : INT ;
   STAT36 : ARRAY  [1 .. 500 ] OF WORD ;
   STAT37 : ARRAY  [1 .. 16 ] OF BYTE ;
   STAT38 : ARRAY  [1 .. 4 ] OF BYTE ;
   STAT39 : ARRAY  [1 .. 16 ] OF BYTE ;
  END_STRUCT ;
BEGIN
   STAT0 := W#16#2717;
   STAT1 := W#16#87;
   STAT2 := W#16#A22;
   STAT3 := W#16#1080;
   STAT4 := W#16#5416;
   STAT5 := W#16#40;
   STAT6 := W#16#0;
   STAT7 := W#16#0;
   STAT8 := W#16#87;
   STAT9 := W#16#2716;
   STAT10 := W#16#2222;
   STAT11 := W#16#8004;
   STAT12 := W#16#1610;
   STAT13 := W#16#6000;
   STAT14 := W#16#0;
   STAT15 := W#16#0;
   STAT16 := 0;
   STAT17 := 4;
   STAT18 := 3;
   STAT19 := 0;
   STAT20[1] := B#16#0;
   STAT20[2] := B#16#0;
   STAT20[3] := B#16#0;
   STAT20[4] := B#16#0;
   STAT20[5] := B#16#0;
   STAT20[6] := B#16#0;
   STAT21[1] := B#16#0;
   STAT21[2] := B#16#0;
   STAT21[3] := B#16#0;
   STAT21[4] := B#16#0;
   STAT21[5] := B#16#0;
   STAT21[6] := B#16#0;
   STAT22[1] := FALSE;
   STAT22[2] := FALSE;
   STAT22[3] := TRUE;
   STAT22[4] := FALSE;
   STAT22[5] := FALSE;
   STAT22[6] := FALSE;
   STAT22[7] := FALSE;
   STAT22[8] := TRUE;
   STAT22[9] := FALSE;
   STAT22[10] := FALSE;
   STAT22[11] := FALSE;
   STAT22[12] := FALSE;
   STAT22[13] := FALSE;
   STAT22[14] := FALSE;
   STAT22[15] := FALSE;
   STAT22[16] := FALSE;
   STAT22[17] := FALSE;
   STAT22[18] := FALSE;
   STAT22[19] := FALSE;
   STAT22[20] := FALSE;
   STAT22[21] := FALSE;
   STAT22[22] := FALSE;
   STAT22[23] := FALSE;
   STAT22[24] := FALSE;
   STAT22[25] := FALSE;
   STAT22[26] := FALSE;
   STAT22[27] := FALSE;
   STAT22[28] := FALSE;
   STAT22[29] := FALSE;
   STAT22[30] := FALSE;
   STAT22[31] := FALSE;
   STAT22[32] := FALSE;
   STAT22[33] := FALSE;
   STAT22[34] := FALSE;
   STAT22[35] := FALSE;
   STAT22[36] := FALSE;
   STAT22[37] := FALSE;
   STAT22[38] := FALSE;
   STAT22[39] := FALSE;
   STAT22[40] := FALSE;
   STAT23[1] := FALSE;
   STAT23[2] := FALSE;
   STAT23[3] := FALSE;
   STAT23[4] := FALSE;
   STAT23[5] := FALSE;
   STAT23[6] := TRUE;
   STAT23[7] := FALSE;
   STAT23[8] := FALSE;
   STAT23[9] := FALSE;
   STAT23[10] := FALSE;
   STAT23[11] := FALSE;
   STAT23[12] := FALSE;
   STAT23[13] := FALSE;
   STAT23[14] := FALSE;
   STAT23[15] := FALSE;
   STAT23[16] := FALSE;
   STAT23[17] := FALSE;
   STAT23[18] := FALSE;
   STAT23[19] := FALSE;
   STAT23[20] := FALSE;
   STAT23[21] := FALSE;
   STAT23[22] := FALSE;
   STAT23[23] := FALSE;
   STAT23[24] := FALSE;
   STAT23[25] := FALSE;
   STAT23[26] := FALSE;
   STAT23[27] := FALSE;
   STAT23[28] := FALSE;
   STAT23[29] := FALSE;
   STAT23[30] := FALSE;
   STAT23[31] := FALSE;
   STAT23[32] := FALSE;
   STAT23[33] := FALSE;
   STAT23[34] := FALSE;
   STAT23[35] := FALSE;
   STAT23[36] := FALSE;
   STAT23[37] := FALSE;
   STAT23[38] := FALSE;
   STAT23[39] := FALSE;
   STAT23[40] := FALSE;
   STAT24 := W#16#400;
   STAT25 := W#16#400;
   STAT26 := W#16#0;
   STAT27 := W#16#0;
   STAT28 := W#16#0;
   STAT29 := W#16#0;
   STAT30 := W#16#0;
   STAT31[1] := W#16#0;
   STAT31[2] := W#16#0;
   STAT31[3] := W#16#0;
   STAT31[4] := W#16#0;
   STAT31[5] := W#16#0;
   STAT31[6] := W#16#0;
   STAT31[7] := W#16#0;
   STAT32 := 100;
   STAT33 := 90;
   STAT34 := 80;
   STAT35 := 0;
   STAT36[1] := W#16#300;
   STAT36[2] := W#16#1418;
   STAT36[3] := W#16#3256;
   STAT36[4] := W#16#B;
   STAT36[5] := W#16#2716;
   STAT36[6] := W#16#200;
   STAT36[7] := W#16#1418;
   STAT36[8] := W#16#3254;
   STAT36[9] := W#16#1;
   STAT36[10] := W#16#2715;
   STAT36[11] := W#16#500;
   STAT36[12] := W#16#1418;
   STAT36[13] := W#16#2636;
   STAT36[14] := W#16#0;
   STAT36[15] := W#16#0;
   STAT36[16] := W#16#400;
   STAT36[17] := W#16#1418;
   STAT36[18] := W#16#2627;
   STAT36[19] := W#16#0;
   STAT36[20] := W#16#2715;
   STAT36[21] := W#16#300;
   STAT36[22] := W#16#1418;
   STAT36[23] := W#16#2556;
   STAT36[24] := W#16#B;
   STAT36[25] := W#16#2715;
   STAT36[26] := W#16#200;
   STAT36[27] := W#16#1418;
   STAT36[28] := W#16#2554;
   STAT36[29] := W#16#1;
   STAT36[30] := W#16#2714;
   STAT36[31] := W#16#500;
   STAT36[32] := W#16#1418;
   STAT36[33] := W#16#2545;
   STAT36[34] := W#16#0;
   STAT36[35] := W#16#0;
   STAT36[36] := W#16#400;
   STAT36[37] := W#16#1418;
   STAT36[38] := W#16#2535;
   STAT36[39] := W#16#0;
   STAT36[40] := W#16#2714;
   STAT36[41] := W#16#300;
   STAT36[42] := W#16#1418;
   STAT36[43] := W#16#2434;
   STAT36[44] := W#16#B;
   STAT36[45] := W#16#2714;
   STAT36[46] := W#16#200;
   STAT36[47] := W#16#1418;
   STAT36[48] := W#16#2432;
   STAT36[49] := W#16#1;
   STAT36[50] := W#16#2713;
   STAT36[51] := W#16#500;
   STAT36[52] := W#16#1418;
   STAT36[53] := W#16#2406;
   STAT36[54] := W#16#0;
   STAT36[55] := W#16#0;
   STAT36[56] := W#16#400;
   STAT36[57] := W#16#1418;
   STAT36[58] := W#16#2356;
   STAT36[59] := W#16#0;
   STAT36[60] := W#16#2713;
   STAT36[61] := W#16#300;
   STAT36[62] := W#16#1418;
   STAT36[63] := W#16#2329;
   STAT36[64] := W#16#B;
   STAT36[65] := W#16#2713;
   STAT36[66] := W#16#200;
   STAT36[67] := W#16#1418;
   STAT36[68] := W#16#2328;
   STAT36[69] := W#16#1;
   STAT36[70] := W#16#2712;
   STAT36[71] := W#16#500;
   STAT36[72] := W#16#1418;
   STAT36[73] := W#16#2318;
   STAT36[74] := W#16#0;
   STAT36[75] := W#16#0;
   STAT36[76] := W#16#400;
   STAT36[77] := W#16#1418;
   STAT36[78] := W#16#2308;
   STAT36[79] := W#16#0;
   STAT36[80] := W#16#2712;
   STAT36[81] := W#16#300;
   STAT36[82] := W#16#1418;
   STAT36[83] := W#16#2112;
   STAT36[84] := W#16#B;
   STAT36[85] := W#16#2712;
   STAT36[86] := W#16#200;
   STAT36[87] := W#16#1418;
   STAT36[88] := W#16#2111;
   STAT36[89] := W#16#1;
   STAT36[90] := W#16#2711;
   STAT36[91] := W#16#500;
   STAT36[92] := W#16#1418;
   STAT36[93] := W#16#2028;
   STAT36[94] := W#16#0;
   STAT36[95] := W#16#0;
   STAT36[96] := W#16#400;
   STAT36[97] := W#16#1418;
   STAT36[98] := W#16#2019;
   STAT36[99] := W#16#0;
   STAT36[100] := W#16#2711;
   STAT36[101] := W#16#300;
   STAT36[102] := W#16#1418;
   STAT36[103] := W#16#1946;
   STAT36[104] := W#16#B;
   STAT36[105] := W#16#2711;
   STAT36[106] := W#16#200;
   STAT36[107] := W#16#1418;
   STAT36[108] := W#16#1945;
   STAT36[109] := W#16#1;
   STAT36[110] := W#16#2710;
   STAT36[111] := W#16#500;
   STAT36[112] := W#16#1418;
   STAT36[113] := W#16#1936;
   STAT36[114] := W#16#0;
   STAT36[115] := W#16#0;
   STAT36[116] := W#16#400;
   STAT36[117] := W#16#1418;
   STAT36[118] := W#16#1926;
   STAT36[119] := W#16#0;
   STAT36[120] := W#16#2710;
   STAT36[121] := W#16#300;
   STAT36[122] := W#16#1418;
   STAT36[123] := W#16#1827;
   STAT36[124] := W#16#B;
   STAT36[125] := W#16#2710;
   STAT36[126] := W#16#200;
   STAT36[127] := W#16#1418;
   STAT36[128] := W#16#1825;
   STAT36[129] := W#16#1;
   STAT36[130] := W#16#2709;
   STAT36[131] := W#16#500;
   STAT36[132] := W#16#1418;
   STAT36[133] := W#16#1758;
   STAT36[134] := W#16#0;
   STAT36[135] := W#16#0;
   STAT36[136] := W#16#400;
   STAT36[137] := W#16#1418;
   STAT36[138] := W#16#1748;
   STAT36[139] := W#16#0;
   STAT36[140] := W#16#2709;
   STAT36[141] := W#16#300;
   STAT36[142] := W#16#1418;
   STAT36[143] := W#16#1722;
   STAT36[144] := W#16#B;
   STAT36[145] := W#16#2709;
   STAT36[146] := W#16#200;
   STAT36[147] := W#16#1418;
   STAT36[148] := W#16#1720;
   STAT36[149] := W#16#1;
   STAT36[150] := W#16#2708;
   STAT36[151] := W#16#500;
   STAT36[152] := W#16#1418;
   STAT36[153] := W#16#1711;
   STAT36[154] := W#16#0;
   STAT36[155] := W#16#0;
   STAT36[156] := W#16#400;
   STAT36[157] := W#16#1418;
   STAT36[158] := W#16#1701;
   STAT36[159] := W#16#0;
   STAT36[160] := W#16#2708;
   STAT36[161] := W#16#300;
   STAT36[162] := W#16#1418;
   STAT36[163] := W#16#1555;
   STAT36[164] := W#16#B;
   STAT36[165] := W#16#2708;
   STAT36[166] := W#16#200;
   STAT36[167] := W#16#1418;
   STAT36[168] := W#16#1553;
   STAT36[169] := W#16#1;
   STAT36[170] := W#16#2707;
   STAT36[171] := W#16#500;
   STAT36[172] := W#16#1418;
   STAT36[173] := W#16#1532;
   STAT36[174] := W#16#0;
   STAT36[175] := W#16#0;
   STAT36[176] := W#16#400;
   STAT36[177] := W#16#1418;
   STAT36[178] := W#16#1522;
   STAT36[179] := W#16#0;
   STAT36[180] := W#16#2707;
   STAT36[181] := W#16#300;
   STAT36[182] := W#16#1418;
   STAT36[183] := W#16#1450;
   STAT36[184] := W#16#B;
   STAT36[185] := W#16#2707;
   STAT36[186] := W#16#200;
   STAT36[187] := W#16#1418;
   STAT36[188] := W#16#1449;
   STAT36[189] := W#16#1;
   STAT36[190] := W#16#2706;
   STAT36[191] := W#16#500;
   STAT36[192] := W#16#1418;
   STAT36[193] := W#16#1425;
   STAT36[194] := W#16#0;
   STAT36[195] := W#16#0;
   STAT36[196] := W#16#400;
   STAT36[197] := W#16#1418;
   STAT36[198] := W#16#1415;
   STAT36[199] := W#16#0;
   STAT36[200] := W#16#2706;
   STAT36[201] := W#16#300;
   STAT36[202] := W#16#1418;
   STAT36[203] := W#16#1346;
   STAT36[204] := W#16#B;
   STAT36[205] := W#16#2706;
   STAT36[206] := W#16#200;
   STAT36[207] := W#16#1418;
   STAT36[208] := W#16#1344;
   STAT36[209] := W#16#1;
   STAT36[210] := W#16#2705;
   STAT36[211] := W#16#500;
   STAT36[212] := W#16#1418;
   STAT36[213] := W#16#1314;
   STAT36[214] := W#16#0;
   STAT36[215] := W#16#0;
   STAT36[216] := W#16#400;
   STAT36[217] := W#16#1418;
   STAT36[218] := W#16#1304;
   STAT36[219] := W#16#0;
   STAT36[220] := W#16#2705;
   STAT36[221] := W#16#300;
   STAT36[222] := W#16#1418;
   STAT36[223] := W#16#1237;
   STAT36[224] := W#16#B;
   STAT36[225] := W#16#2705;
   STAT36[226] := W#16#200;
   STAT36[227] := W#16#1418;
   STAT36[228] := W#16#1236;
   STAT36[229] := W#16#1;
   STAT36[230] := W#16#2704;
   STAT36[231] := W#16#500;
   STAT36[232] := W#16#1418;
   STAT36[233] := W#16#1227;
   STAT36[234] := W#16#0;
   STAT36[235] := W#16#0;
   STAT36[236] := W#16#400;
   STAT36[237] := W#16#1418;
   STAT36[238] := W#16#1217;
   STAT36[239] := W#16#0;
   STAT36[240] := W#16#2704;
   STAT36[241] := W#16#300;
   STAT36[242] := W#16#1418;
   STAT36[243] := W#16#1029;
   STAT36[244] := W#16#B;
   STAT36[245] := W#16#2704;
   STAT36[246] := W#16#200;
   STAT36[247] := W#16#1418;
   STAT36[248] := W#16#1028;
   STAT36[249] := W#16#1;
   STAT36[250] := W#16#2703;
   STAT36[251] := W#16#500;
   STAT36[252] := W#16#1418;
   STAT36[253] := W#16#1012;
   STAT36[254] := W#16#0;
   STAT36[255] := W#16#0;
   STAT36[256] := W#16#400;
   STAT36[257] := W#16#1418;
   STAT36[258] := W#16#1003;
   STAT36[259] := W#16#0;
   STAT36[260] := W#16#2703;
   STAT36[261] := W#16#300;
   STAT36[262] := W#16#1418;
   STAT36[263] := W#16#917;
   STAT36[264] := W#16#B;
   STAT36[265] := W#16#2703;
   STAT36[266] := W#16#200;
   STAT36[267] := W#16#1418;
   STAT36[268] := W#16#915;
   STAT36[269] := W#16#1;
   STAT36[270] := W#16#2702;
   STAT36[271] := W#16#500;
   STAT36[272] := W#16#1418;
   STAT36[273] := W#16#846;
   STAT36[274] := W#16#0;
   STAT36[275] := W#16#0;
   STAT36[276] := W#16#400;
   STAT36[277] := W#16#1418;
   STAT36[278] := W#16#837;
   STAT36[279] := W#16#0;
   STAT36[280] := W#16#2702;
   STAT36[281] := W#16#300;
   STAT36[282] := W#16#1418;
   STAT36[283] := W#16#802;
   STAT36[284] := W#16#B;
   STAT36[285] := W#16#2702;
   STAT36[286] := W#16#200;
   STAT36[287] := W#16#1418;
   STAT36[288] := W#16#801;
   STAT36[289] := W#16#1;
   STAT36[290] := W#16#2701;
   STAT36[291] := W#16#500;
   STAT36[292] := W#16#1418;
   STAT36[293] := W#16#509;
   STAT36[294] := W#16#0;
   STAT36[295] := W#16#0;
   STAT36[296] := W#16#400;
   STAT36[297] := W#16#1418;
   STAT36[298] := W#16#459;
   STAT36[299] := W#16#0;
   STAT36[300] := W#16#2701;
   STAT36[301] := W#16#300;
   STAT36[302] := W#16#1418;
   STAT36[303] := W#16#415;
   STAT36[304] := W#16#B;
   STAT36[305] := W#16#2701;
   STAT36[306] := W#16#200;
   STAT36[307] := W#16#1418;
   STAT36[308] := W#16#413;
   STAT36[309] := W#16#1;
   STAT36[310] := W#16#2700;
   STAT36[311] := W#16#500;
   STAT36[312] := W#16#1418;
   STAT36[313] := W#16#404;
   STAT36[314] := W#16#0;
   STAT36[315] := W#16#0;
   STAT36[316] := W#16#400;
   STAT36[317] := W#16#1418;
   STAT36[318] := W#16#354;
   STAT36[319] := W#16#0;
   STAT36[320] := W#16#2700;
   STAT36[321] := W#16#300;
   STAT36[322] := W#16#1418;
   STAT36[323] := W#16#306;
   STAT36[324] := W#16#B;
   STAT36[325] := W#16#2700;
   STAT36[326] := W#16#200;
   STAT36[327] := W#16#1418;
   STAT36[328] := W#16#303;
   STAT36[329] := W#16#1;
   STAT36[330] := W#16#2699;
   STAT36[331] := W#16#500;
   STAT36[332] := W#16#1418;
   STAT36[333] := W#16#207;
   STAT36[334] := W#16#0;
   STAT36[335] := W#16#0;
   STAT36[336] := W#16#400;
   STAT36[337] := W#16#1418;
   STAT36[338] := W#16#157;
   STAT36[339] := W#16#0;
   STAT36[340] := W#16#2699;
   STAT36[341] := W#16#300;
   STAT36[342] := W#16#1418;
   STAT36[343] := W#16#127;
   STAT36[344] := W#16#B;
   STAT36[345] := W#16#2699;
   STAT36[346] := W#16#200;
   STAT36[347] := W#16#1418;
   STAT36[348] := W#16#126;
   STAT36[349] := W#16#1;
   STAT36[350] := W#16#2698;
   STAT36[351] := W#16#500;
   STAT36[352] := W#16#1418;
   STAT36[353] := W#16#52;
   STAT36[354] := W#16#0;
   STAT36[355] := W#16#0;
   STAT36[356] := W#16#400;
   STAT36[357] := W#16#1418;
   STAT36[358] := W#16#42;
   STAT36[359] := W#16#0;
   STAT36[360] := W#16#2698;
   STAT36[361] := W#16#300;
   STAT36[362] := W#16#1418;
   STAT36[363] := W#16#11;
   STAT36[364] := W#16#B;
   STAT36[365] := W#16#2698;
   STAT36[366] := W#16#200;
   STAT36[367] := W#16#1418;
   STAT36[368] := W#16#9;
   STAT36[369] := W#16#1;
   STAT36[370] := W#16#2697;
   STAT36[371] := W#16#500;
   STAT36[372] := W#16#1417;
   STAT36[373] := W#16#5939;
   STAT36[374] := W#16#0;
   STAT36[375] := W#16#0;
   STAT36[376] := W#16#400;
   STAT36[377] := W#16#1417;
   STAT36[378] := W#16#5929;
   STAT36[379] := W#16#0;
   STAT36[380] := W#16#2697;
   STAT36[381] := W#16#300;
   STAT36[382] := W#16#1417;
   STAT36[383] := W#16#5900;
   STAT36[384] := W#16#B;
   STAT36[385] := W#16#2697;
   STAT36[386] := W#16#200;
   STAT36[387] := W#16#1417;
   STAT36[388] := W#16#5858;
   STAT36[389] := W#16#1;
   STAT36[390] := W#16#2696;
   STAT36[391] := W#16#500;
   STAT36[392] := W#16#1417;
   STAT36[393] := W#16#5832;
   STAT36[394] := W#16#0;
   STAT36[395] := W#16#0;
   STAT36[396] := W#16#400;
   STAT36[397] := W#16#1417;
   STAT36[398] := W#16#5822;
   STAT36[399] := W#16#0;
   STAT36[400] := W#16#2696;
   STAT36[401] := W#16#300;
   STAT36[402] := W#16#1417;
   STAT36[403] := W#16#5748;
   STAT36[404] := W#16#B;
   STAT36[405] := W#16#2696;
   STAT36[406] := W#16#200;
   STAT36[407] := W#16#1417;
   STAT36[408] := W#16#5746;
   STAT36[409] := W#16#1;
   STAT36[410] := W#16#2695;
   STAT36[411] := W#16#500;
   STAT36[412] := W#16#1417;
   STAT36[413] := W#16#5713;
   STAT36[414] := W#16#0;
   STAT36[415] := W#16#0;
   STAT36[416] := W#16#400;
   STAT36[417] := W#16#1417;
   STAT36[418] := W#16#5703;
   STAT36[419] := W#16#0;
   STAT36[420] := W#16#2695;
   STAT36[421] := W#16#300;
   STAT36[422] := W#16#1417;
   STAT36[423] := W#16#5635;
   STAT36[424] := W#16#B;
   STAT36[425] := W#16#2695;
   STAT36[426] := W#16#200;
   STAT36[427] := W#16#1417;
   STAT36[428] := W#16#5633;
   STAT36[429] := W#16#1;
   STAT36[430] := W#16#2694;
   STAT36[431] := W#16#500;
   STAT36[432] := W#16#1417;
   STAT36[433] := W#16#5606;
   STAT36[434] := W#16#0;
   STAT36[435] := W#16#0;
   STAT36[436] := W#16#400;
   STAT36[437] := W#16#1417;
   STAT36[438] := W#16#5556;
   STAT36[439] := W#16#0;
   STAT36[440] := W#16#2694;
   STAT36[441] := W#16#300;
   STAT36[442] := W#16#1417;
   STAT36[443] := W#16#5520;
   STAT36[444] := W#16#B;
   STAT36[445] := W#16#2694;
   STAT36[446] := W#16#200;
   STAT36[447] := W#16#1417;
   STAT36[448] := W#16#5519;
   STAT36[449] := W#16#1;
   STAT36[450] := W#16#2693;
   STAT36[451] := W#16#500;
   STAT36[452] := W#16#1417;
   STAT36[453] := W#16#5442;
   STAT36[454] := W#16#0;
   STAT36[455] := W#16#0;
   STAT36[456] := W#16#400;
   STAT36[457] := W#16#1417;
   STAT36[458] := W#16#5432;
   STAT36[459] := W#16#0;
   STAT36[460] := W#16#2693;
   STAT36[461] := W#16#300;
   STAT36[462] := W#16#1417;
   STAT36[463] := W#16#5406;
   STAT36[464] := W#16#B;
   STAT36[465] := W#16#2693;
   STAT36[466] := W#16#200;
   STAT36[467] := W#16#1417;
   STAT36[468] := W#16#5404;
   STAT36[469] := W#16#1;
   STAT36[470] := W#16#2692;
   STAT36[471] := W#16#500;
   STAT36[472] := W#16#1417;
   STAT36[473] := W#16#5324;
   STAT36[474] := W#16#0;
   STAT36[475] := W#16#0;
   STAT36[476] := W#16#400;
   STAT36[477] := W#16#1417;
   STAT36[478] := W#16#5315;
   STAT36[479] := W#16#0;
   STAT36[480] := W#16#2692;
   STAT36[481] := W#16#300;
   STAT36[482] := W#16#1417;
   STAT36[483] := W#16#5249;
   STAT36[484] := W#16#B;
   STAT36[485] := W#16#2692;
   STAT36[486] := W#16#200;
   STAT36[487] := W#16#1417;
   STAT36[488] := W#16#5248;
   STAT36[489] := W#16#1;
   STAT36[490] := W#16#2691;
   STAT36[491] := W#16#500;
   STAT36[492] := W#16#1417;
   STAT36[493] := W#16#5217;
   STAT36[494] := W#16#0;
   STAT36[495] := W#16#0;
   STAT36[496] := W#16#400;
   STAT36[497] := W#16#1417;
   STAT36[498] := W#16#5208;
   STAT36[499] := W#16#0;
   STAT36[500] := W#16#2691;
   STAT37[1] := B#16#0;
   STAT37[2] := B#16#87;
   STAT37[3] := B#16#27;
   STAT37[4] := B#16#16;
   STAT37[5] := B#16#22;
   STAT37[6] := B#16#22;
   STAT37[7] := B#16#80;
   STAT37[8] := B#16#4;
   STAT37[9] := B#16#16;
   STAT37[10] := B#16#10;
   STAT37[11] := B#16#60;
   STAT37[12] := B#16#0;
   STAT37[13] := B#16#0;
   STAT37[14] := B#16#0;
   STAT37[15] := B#16#0;
   STAT37[16] := B#16#0;
   STAT38[1] := B#16#0;
   STAT38[2] := B#16#0;
   STAT38[3] := B#16#0;
   STAT38[4] := B#16#0;
   STAT39[1] := B#16#27;
   STAT39[2] := B#16#16;
   STAT39[3] := B#16#0;
   STAT39[4] := B#16#87;
   STAT39[5] := B#16#22;
   STAT39[6] := B#16#22;
   STAT39[7] := B#16#4;
   STAT39[8] := B#16#80;
   STAT39[9] := B#16#10;
   STAT39[10] := B#16#16;
   STAT39[11] := B#16#0;
   STAT39[12] := B#16#60;
   STAT39[13] := B#16#0;
   STAT39[14] := B#16#0;
   STAT39[15] := B#16#0;
   STAT39[16] := B#16#0;
END_DATA_BLOCK

DATA_BLOCK DB 168
VERSION : 0.1


